LIN {X 0,Y 385.624,Z 461.843,A -85,B 0,C 180,E1 17447.458,E2 17447.458} C_VEL
LIN {X 0,Y 393.74,Z 473.597,A -85,B 0,C 180,E1 17445.289,E2 17445.289} C_VEL
LIN {X 0,Y 402.693,Z 487.716,A -85,B 0,C 180,E1 17443.13,E2 17443.13} C_VEL
LIN {X 0,Y 410.584,Z 501.659,A -85,B 0,C 180,E1 17441.371,E2 17441.371} C_VEL
LIN {X 0,Y 399.515,Z 724.653,A -85,B 0,C 180,E1 17436.869,E2 17436.869} C_VEL
LIN {X 0,Y 397.719,Z 745.499,A -85,B 0,C 180,E1 17436.196,E2 17436.196} C_VEL
LIN {X 0,Y 395.346,Z 765.584,A -85,B 0,C 180,E1 17435.296,E2 17435.296} C_VEL
LIN {X 0,Y 392.457,Z 785.369,A -85,B 0,C 180,E1 17434.136,E2 17434.136} C_VEL
LIN {X 0,Y 389.149,Z 804.356,A -85,B 0,C 180,E1 17432.737,E2 17432.737} C_VEL
LIN {X 0,Y 385.5,Z 822.639,A -85,B 0,C 180,E1 17431.079,E2 17431.079} C_VEL
LIN {X 0,Y 381.768,Z 839.649,A -85,B 0,C 180,E1 17429.2,E2 17429.2} C_VEL
LIN {X 0,Y 378.016,Z 855.337,A -85,B 0,C 180,E1 17427.11,E2 17427.11} C_VEL
LIN {X 0,Y 374.362,Z 870.021,A -85,B 0,C 180,E1 17424.767,E2 17424.767} C_VEL
LIN {X 0,Y 370.795,Z 884.125,A -85,B 0,C 180,E1 17422.061,E2 17422.061} C_VEL
LIN {X 0,Y 367.789,Z 896.136,A -85,B 0,C 180,E1 17419.272,E2 17419.272} C_VEL
LIN {X 0,Y 365.351,Z 906.362,A -85,B 0,C 180,E1 17416.397,E2 17416.397} C_VEL
LIN {X 0,Y 363.362,Z 915.457,A -85,B 0,C 180,E1 17413.243,E2 17413.243} C_VEL
LIN {X 0,Y 361.969,Z 922.647,A -85,B 0,C 180,E1 17410.056,E2 17410.056} C_VEL
LIN {X 0,Y 361.097,Z 928.123,A -85,B 0,C 180,E1 17406.848,E2 17406.848} C_VEL
LIN {X 0,Y 360.609,Z 932.126,A -85,B 0,C 180,E1 17403.483,E2 17403.483} C_VEL
LIN {X 0,Y 360.394,Z 934.36,A -85,B 0,C 180,E1 17400.322,E2 17400.322} C_VEL
LIN {X 0,Y 360.332,Z 935.093,A -85,B 0,C 180,E1 17397.243,E2 17397.243} C_VEL
LIN {X 0,Y 360.36,Z 934.348,A -85,B 0,C 180,E1 17394.066,E2 17394.066} C_VEL
LIN {X 0,Y 360.529,Z 932.047,A -85,B 0,C 180,E1 17390.788,E2 17390.788} C_VEL
LIN {X 0,Y 360.933,Z 928.226,A -85,B 0,C 180,E1 17387.571,E2 17387.571} C_VEL
LIN {X 0,Y 361.721,Z 922.518,A -85,B 0,C 180,E1 17384.238,E2 17384.238} C_VEL
LIN {X 0,Y 363.027,Z 914.958,A -85,B 0,C 180,E1 17380.951,E2 17380.951} C_VEL
LIN {X 0,Y 364.829,Z 905.967,A -85,B 0,C 180,E1 17377.872,E2 17377.872} C_VEL
LIN {X 0,Y 365.782,Z 901.545,A -85,B 0,C 180,E1 17376.571,E2 17376.571} C_VEL
LIN {X 0,Y 365.685,Z 897.934,A -85,B 0,C 180,E1 17375.494,E2 17375.494} C_VEL
LIN {X 0,Y 362.411,Z 888.671,A -85,B 0,C 180,E1 17372.727,E2 17372.727} C_VEL
LIN {X 0,Y 362.563,Z 884.364,A -85,B 0,C 180,E1 17371.705,E2 17371.705} C_VEL
LIN {X 0,Y 365.958,Z 870.807,A -85,B 0,C 180,E1 17369.057,E2 17369.057} C_VEL
LIN {X 0,Y 369.577,Z 856.128,A -85,B 0,C 180,E1 17366.665,E2 17366.665} C_VEL
LIN {X 0,Y 373.549,Z 839.227,A -85,B 0,C 180,E1 17364.39,E2 17364.39} C_VEL
LIN {X 0,Y 377.305,Z 821.832,A -85,B 0,C 180,E1 17362.459,E2 17362.459} C_VEL
LIN {X 0,Y 380.805,Z 804.113,A -85,B 0,C 180,E1 17360.841,E2 17360.841} C_VEL
LIN {X 0,Y 384.175,Z 784.574,A -85,B 0,C 180,E1 17359.386,E2 17359.386} C_VEL
LIN {X 0,Y 387.031,Z 764.817,A -85,B 0,C 180,E1 17358.221,E2 17358.221} C_VEL
LIN {X 0,Y 389.427,Z 744.323,A -85,B 0,C 180,E1 17357.301,E2 17357.301} C_VEL
LIN {X 0,Y 391.197,Z 723.212,A -85,B 0,C 180,E1 17356.623,E2 17356.623} C_VEL
LIN {X 0,Y 394.489,Z 650.13,A -85,B 0,C 180,E1 17355.144,E2 17355.144} C_VEL
LIN {X 0,Y 401.065,Z 502.372,A -85,B 0,C 180,E1 17352.239,E2 17352.239} C_VEL
LIN {X 0,Y 390.659,Z 484.683,A -85,B 0,C 180,E1 17350.151,E2 17350.151} C_VEL
LIN {X 0,Y 380.819,Z 469.313,A -85,B 0,C 180,E1 17348.046,E2 17348.046} C_VEL
LIN {X 0,Y 369.494,Z 452.63,A -85,B 0,C 180,E1 17345.369,E2 17345.369} C_VEL
LIN {X 0,Y 363.337,Z 440.093,A -85,B 0,C 180,E1 17342.05,E2 17342.05} C_VEL
LIN {X 0,Y 360.294,Z 434.531,A -85,B 0,C 180,E1 17340.395,E2 17340.395} C_VEL
LIN {X 0,Y 358.363,Z 430.7,A -85,B 0,C 180,E1 17339.244,E2 17339.244} C_VEL
LIN {X 0,Y 356.284,Z 426.499,A -85,B 0,C 180,E1 17337.944,E2 17337.944} C_VEL
LIN {X 0,Y 354.253,Z 423.304,A -85,B 0,C 180,E1 17336.798,E2 17336.798} C_VEL
LIN {X 0,Y 353.891,Z 421.837,A -85,B 0,C 180,E1 17336.274,E2 17336.274} C_VEL
LIN {X 0,Y 353.868,Z 421.638,A -85,B 0,C 180,E1 17332.029,E2 17332.029} C_VEL
LIN {X 0,Y 353.865,Z 421.638,A -85,B 0,C 180,E1 17327.738,E2 17327.738} C_VEL
LIN {X 0,Y 353.864,Z 421.647,A -85,B 0,C 180,E1 17323.431,E2 17323.431} C_VEL
LIN {X 0,Y 353.871,Z 421.657,A -85,B 0,C 180,E1 17319.266,E2 17319.266} C_VEL
LIN {X 0,Y 353.861,Z 421.644,A -85,B 0,C 180,E1 17314.97,E2 17314.97} C_VEL
LIN {X 0,Y 353.86,Z 421.627,A -85,B 0,C 180,E1 17310.76,E2 17310.76} C_VEL
LIN {X 0,Y 353.862,Z 421.627,A -85,B 0,C 180,E1 17306.697,E2 17306.697} C_VEL
LIN {X 0,Y 353.865,Z 421.651,A -85,B 0,C 180,E1 17302.424,E2 17302.424} C_VEL
LIN {X 0,Y 353.863,Z 421.647,A -85,B 0,C 180,E1 17298.109,E2 17298.109} C_VEL
LIN {X 0,Y 353.86,Z 421.626,A -85,B 0,C 180,E1 17293.897,E2 17293.897} C_VEL
LIN {X 0,Y 353.86,Z 421.63,A -85,B 0,C 180,E1 17289.761,E2 17289.761} C_VEL
LIN {X 0,Y 353.863,Z 421.653,A -85,B 0,C 180,E1 17285.513,E2 17285.513} C_VEL
LIN {X 0,Y 353.866,Z 421.645,A -85,B 0,C 180,E1 17281.296,E2 17281.296} C_VEL
LIN {X 0,Y 353.86,Z 421.629,A -85,B 0,C 180,E1 17277.085,E2 17277.085} C_VEL
LIN {X 0,Y 353.87,Z 421.625,A -85,B 0,C 180,E1 17272.859,E2 17272.859} C_VEL
LIN {X 0,Y 353.862,Z 421.633,A -85,B 0,C 180,E1 17268.593,E2 17268.593} C_VEL
LIN {X 0,Y 353.867,Z 421.64,A -85,B 0,C 180,E1 17264.43,E2 17264.43} C_VEL
LIN {X 0,Y 353.863,Z 421.642,A -85,B 0,C 180,E1 17260.181,E2 17260.181} C_VEL
LIN {X 0,Y 353.907,Z 421.916,A -85,B 0,C 180,E1 17256.647,E2 17256.647} C_VEL
LIN {X 0,Y 355.277,Z 425.289,A -85,B 0,C 180,E1 17255.563,E2 17255.563} C_VEL
LIN {X 0,Y 356.837,Z 427.334,A -85,B 0,C 180,E1 17254.793,E2 17254.793} C_VEL
LIN {X 0,Y 358.714,Z 431.017,A -85,B 0,C 180,E1 17253.693,E2 17253.693} C_VEL
LIN {X 0,Y 359.897,Z 433.003,A -85,B 0,C 180,E1 17253.074,E2 17253.074} C_VEL
LIN {X 0,Y 362.824,Z 438.361,A -85,B 0,C 180,E1 17251.527,E2 17251.527} C_VEL
LIN {X 0,Y 367.452,Z 446.794,A -85,B 0,C 180,E1 17249.233,E2 17249.233} C_VEL
LIN {X 0,Y 371.993,Z 455.21,A -85,B 0,C 180,E1 17247.208,E2 17247.208} C_VEL
LIN {X 0,Y 385.078,Z 473.968,A -85,B 0,C 180,E1 17244.207,E2 17244.207} C_VEL
LIN {X 0,Y 396.972,Z 492.362,A -85,B 0,C 180,E1 17241.713,E2 17241.713} C_VEL
LIN {X 0,Y 405.843,Z 507.315,A -85,B 0,C 180,E1 17239.976,E2 17239.976} C_VEL
LIN {X 0,Y 396.961,Z 726.559,A -85,B 0,C 180,E1 17235.789,E2 17235.789} C_VEL
LIN {X 0,Y 395.432,Z 758.529,A -85,B 0,C 180,E1 17235.13,E2 17235.13} C_VEL
LIN {X 0,Y 393.317,Z 780.529,A -85,B 0,C 180,E1 17234.471,E2 17234.471} C_VEL
LIN {X 0,Y 390.557,Z 801.649,A -85,B 0,C 180,E1 17233.573,E2 17233.573} C_VEL
LIN {X 0,Y 387.183,Z 823.142,A -85,B 0,C 180,E1 17232.379,E2 17232.379} C_VEL
LIN {X 0,Y 383.567,Z 842.972,A -85,B 0,C 180,E1 17231,E2 17231} C_VEL
LIN {X 0,Y 379.663,Z 861.754,A -85,B 0,C 180,E1 17229.399,E2 17229.399} C_VEL
LIN {X 0,Y 375.513,Z 880.297,A -85,B 0,C 180,E1 17227.49,E2 17227.49} C_VEL
LIN {X 0,Y 371.385,Z 897.84,A -85,B 0,C 180,E1 17225.339,E2 17225.339} C_VEL
LIN {X 0,Y 367.337,Z 914.388,A -85,B 0,C 180,E1 17222.927,E2 17222.927} C_VEL
LIN {X 0,Y 363.625,Z 929.506,A -85,B 0,C 180,E1 17220.3,E2 17220.3} C_VEL
LIN {X 0,Y 360.131,Z 944.253,A -85,B 0,C 180,E1 17217.268,E2 17217.268} C_VEL
LIN {X 0,Y 357.383,Z 956.769,A -85,B 0,C 180,E1 17214.21,E2 17214.21} C_VEL
LIN {X 0,Y 355.303,Z 967.347,A -85,B 0,C 180,E1 17211.116,E2 17211.116} C_VEL
LIN {X 0,Y 353.742,Z 976.8,A -85,B 0,C 180,E1 17207.777,E2 17207.777} C_VEL
LIN {X 0,Y 352.792,Z 984.497,A -85,B 0,C 180,E1 17204.445,E2 17204.445} C_VEL
LIN {X 0,Y 352.315,Z 990.433,A -85,B 0,C 180,E1 17201.13,E2 17201.13} C_VEL
LIN {X 0,Y 352.13,Z 994.962,A -85,B 0,C 180,E1 17197.673,E2 17197.673} C_VEL
LIN {X 0,Y 352.135,Z 997.53,A -85,B 0,C 180,E1 17194.706,E2 17194.706} C_VEL
LIN {X 0,Y 352.185,Z 998.914,A -85,B 0,C 180,E1 17191.305,E2 17191.305} C_VEL
LIN {X 0,Y 352.184,Z 998.823,A -85,B 0,C 180,E1 17188.377,E2 17188.377} C_VEL
LIN {X 0,Y 352.141,Z 997.271,A -85,B 0,C 180,E1 17185.117,E2 17185.117} C_VEL
LIN {X 0,Y 352.148,Z 994.589,A -85,B 0,C 180,E1 17182.171,E2 17182.171} C_VEL
LIN {X 0,Y 352.34,Z 989.877,A -85,B 0,C 180,E1 17178.712,E2 17178.712} C_VEL
LIN {X 0,Y 352.825,Z 983.792,A -85,B 0,C 180,E1 17175.395,E2 17175.395} C_VEL
LIN {X 0,Y 353.789,Z 975.895,A -85,B 0,C 180,E1 17172.062,E2 17172.062} C_VEL
LIN {X 0,Y 355.462,Z 965.704,A -85,B 0,C 180,E1 17168.556,E2 17168.556} C_VEL
LIN {X 0,Y 357.648,Z 954.623,A -85,B 0,C 180,E1 17165.388,E2 17165.388} C_VEL
LIN {X 0,Y 360.561,Z 941.345,A -85,B 0,C 180,E1 17162.238,E2 17162.238} C_VEL
LIN {X 0,Y 363.858,Z 927.441,A -85,B 0,C 180,E1 17159.45,E2 17159.45} C_VEL
LIN {X 0,Y 367.695,Z 911.791,A -85,B 0,C 180,E1 17156.78,E2 17156.78} C_VEL
LIN {X 0,Y 371.908,Z 894.648,A -85,B 0,C 180,E1 17154.316,E2 17154.316} C_VEL
LIN {X 0,Y 376.215,Z 876.414,A -85,B 0,C 180,E1 17152.132,E2 17152.132} C_VEL
LIN {X 0,Y 380.472,Z 857.446,A -85,B 0,C 180,E1 17150.236,E2 17150.236} C_VEL
LIN {X 0,Y 384.412,Z 838.439,A -85,B 0,C 180,E1 17148.656,E2 17148.656} C_VEL
LIN {X 0,Y 387.995,Z 818.936,A -85,B 0,C 180,E1 17147.338,E2 17147.338} C_VEL
LIN {X 0,Y 391.235,Z 798.45,A -85,B 0,C 180,E1 17146.233,E2 17146.233} C_VEL
LIN {X 0,Y 394.042,Z 777.211,A -85,B 0,C 180,E1 17145.357,E2 17145.357} C_VEL
LIN {X 0,Y 396.122,Z 755.661,A -85,B 0,C 180,E1 17144.721,E2 17144.721} C_VEL
LIN {X 0,Y 397.895,Z 717.515,A -85,B 0,C 180,E1 17143.948,E2 17143.948} C_VEL
LIN {X 0,Y 406.806,Z 512.285,A -85,B 0,C 180,E1 17139.967,E2 17139.967} C_VEL
LIN {X 0,Y 406.945,Z 506.851,A -85,B 0,C 180,E1 17139.84,E2 17139.84} C_VEL
LIN {X 0,Y 398.811,Z 492.533,A -85,B 0,C 180,E1 17138.01,E2 17138.01} C_VEL
LIN {X 0,Y 390.411,Z 479.057,A -85,B 0,C 180,E1 17135.952,E2 17135.952} C_VEL
LIN {X 0,Y 381.877,Z 466.595,A -85,B 0,C 180,E1 17133.625,E2 17133.625} C_VEL
LIN {X 0,Y 374.629,Z 456.983,A -85,B 0,C 180,E1 17131.406,E2 17131.406} C_VEL
LIN {X 0,Y 372.382,Z 453.459,A -85,B 0,C 180,E1 17130.495,E2 17130.495} C_VEL
LIN {X 0,Y 369.247,Z 447.902,A -85,B 0,C 180,E1 17128.462,E2 17128.462} C_VEL
LIN {X 0,Y 366.715,Z 443.261,A -85,B 0,C 180,E1 17126.56,E2 17126.56} C_VEL
LIN {X 0,Y 364.44,Z 439.225,A -85,B 0,C 180,E1 17124.646,E2 17124.646} C_VEL
LIN {X 0,Y 361.343,Z 434.166,A -85,B 0,C 180,E1 17121.593,E2 17121.593} C_VEL
LIN {X 0,Y 360.702,Z 432.95,A -85,B 0,C 180,E1 17120.782,E2 17120.782} C_VEL
LIN {X 0,Y 357.518,Z 427.654,A -85,B 0,C 180,E1 17115.075,E2 17115.075} C_VEL
LIN {X 0,Y 356.711,Z 426.904,A -85,B 0,C 180,E1 17110.988,E2 17110.988} C_VEL
LIN {X 0,Y 357.579,Z 427.797,A -85,B 0,C 180,E1 17106.905,E2 17106.905} C_VEL
LIN {X 0,Y 361.007,Z 433.575,A -85,B 0,C 180,E1 17100.952,E2 17100.952} C_VEL
LIN {X 0,Y 363.131,Z 437.618,A -85,B 0,C 180,E1 17098.422,E2 17098.422} C_VEL
LIN {X 0,Y 364.003,Z 438.907,A -85,B 0,C 180,E1 17097.638,E2 17097.638} C_VEL
LIN {X 0,Y 366.024,Z 442.707,A -85,B 0,C 180,E1 17095.77,E2 17095.77} C_VEL
LIN {X 0,Y 366.893,Z 444.481,A -85,B 0,C 180,E1 17094.997,E2 17094.997} C_VEL
LIN {X 0,Y 369.261,Z 448.859,A -85,B 0,C 180,E1 17093.157,E2 17093.157} C_VEL
LIN {X 0,Y 371.755,Z 453.713,A -85,B 0,C 180,E1 17091.415,E2 17091.415} C_VEL
LIN {X 0,Y 378.963,Z 463.457,A -85,B 0,C 180,E1 17089.01,E2 17089.01} C_VEL
LIN {X 0,Y 385.61,Z 472.854,A -85,B 0,C 180,E1 17087.061,E2 17087.061} C_VEL
LIN {X 0,Y 394.091,Z 485.886,A -85,B 0,C 180,E1 17084.813,E2 17084.813} C_VEL
LIN {X 0,Y 402.845,Z 500.747,A -85,B 0,C 180,E1 17082.709,E2 17082.709} C_VEL
LIN {X 0,Y 405.224,Z 505.329,A -85,B 0,C 180,E1 17082.16,E2 17082.16} C_VEL
LIN {X 0,Y 393.777,Z 725.022,A -85,B 0,C 180,E1 17077.674,E2 17077.674} C_VEL
LIN {X 0,Y 391.902,Z 745.893,A -85,B 0,C 180,E1 17076.993,E2 17076.993} C_VEL
LIN {X 0,Y 389.528,Z 765.225,A -85,B 0,C 180,E1 17076.123,E2 17076.123} C_VEL
LIN {X 0,Y 386.385,Z 785.898,A -85,B 0,C 180,E1 17074.907,E2 17074.907} C_VEL
LIN {X 0,Y 383.048,Z 804.359,A -85,B 0,C 180,E1 17073.539,E2 17073.539} C_VEL
LIN {X 0,Y 379.303,Z 822.416,A -85,B 0,C 180,E1 17071.898,E2 17071.898} C_VEL
LIN {X 0,Y 375.129,Z 840.491,A -85,B 0,C 180,E1 17069.878,E2 17069.878} C_VEL
LIN {X 0,Y 371.183,Z 856.196,A -85,B 0,C 180,E1 17067.751,E2 17067.751} C_VEL
LIN {X 0,Y 367.371,Z 870.732,A -85,B 0,C 180,E1 17065.394,E2 17065.394} C_VEL
LIN {X 0,Y 363.788,Z 884.115,A -85,B 0,C 180,E1 17062.795,E2 17062.795} C_VEL
LIN {X 0,Y 360.755,Z 895.549,A -85,B 0,C 180,E1 17060.143,E2 17060.143} C_VEL
LIN {X 0,Y 357.936,Z 906.576,A -85,B 0,C 180,E1 17057.031,E2 17057.031} C_VEL
LIN {X 0,Y 355.716,Z 915.92,A -85,B 0,C 180,E1 17053.74,E2 17053.74} C_VEL
LIN {X 0,Y 354.193,Z 923.167,A -85,B 0,C 180,E1 17050.481,E2 17050.481} C_VEL
LIN {X 0,Y 353.242,Z 928.592,A -85,B 0,C 180,E1 17047.276,E2 17047.276} C_VEL
LIN {X 0,Y 352.704,Z 932.594,A -85,B 0,C 180,E1 17043.944,E2 17043.944} C_VEL
LIN {X 0,Y 352.451,Z 934.981,A -85,B 0,C 180,E1 17040.701,E2 17040.701} C_VEL
LIN {X 0,Y 352.365,Z 935.784,A -85,B 0,C 180,E1 17037.545,E2 17037.545} C_VEL
LIN {X 0,Y 352.39,Z 935.18,A -85,B 0,C 180,E1 17034.289,E2 17034.289} C_VEL
LIN {X 0,Y 352.54,Z 933.159,A -85,B 0,C 180,E1 17031.076,E2 17031.076} C_VEL
LIN {X 0,Y 352.941,Z 929.545,A -85,B 0,C 180,E1 17027.812,E2 17027.812} C_VEL
LIN {X 0,Y 353.672,Z 924.319,A -85,B 0,C 180,E1 17024.569,E2 17024.569} C_VEL
LIN {X 0,Y 354.901,Z 917.473,A -85,B 0,C 180,E1 17021.356,E2 17021.356} C_VEL
LIN {X 0,Y 356.67,Z 908.995,A -85,B 0,C 180,E1 17018.216,E2 17018.216} C_VEL
LIN {X 0,Y 358.942,Z 899.215,A -85,B 0,C 180,E1 17015.271,E2 17015.271} C_VEL
LIN {X 0,Y 361.991,Z 886.756,A -85,B 0,C 180,E1 17012.213,E2 17012.213} C_VEL
LIN {X 0,Y 362.563,Z 884.364,A -85,B 0,C 180,E1 17011.705,E2 17011.705} C_VEL
LIN {X 0,Y 362.794,Z 879.981,A -85,B 0,C 180,E1 17010.698,E2 17010.698} C_VEL
LIN {X 0,Y 360.416,Z 868.807,A -85,B 0,C 180,E1 17008.065,E2 17008.065} C_VEL
LIN {X 0,Y 360.833,Z 863.748,A -85,B 0,C 180,E1 17007.134,E2 17007.134} C_VEL
LIN {X 0,Y 364.759,Z 848.234,A -85,B 0,C 180,E1 17004.807,E2 17004.807} C_VEL
LIN {X 0,Y 368.832,Z 831.005,A -85,B 0,C 180,E1 17002.677,E2 17002.677} C_VEL
LIN {X 0,Y 372.614,Z 813.432,A -85,B 0,C 180,E1 17000.888,E2 17000.888} C_VEL
LIN {X 0,Y 376.151,Z 795.04,A -85,B 0,C 180,E1 16999.351,E2 16999.351} C_VEL
LIN {X 0,Y 379.348,Z 775.813,A -85,B 0,C 180,E1 16998.056,E2 16998.056} C_VEL
LIN {X 0,Y 382.057,Z 756.052,A -85,B 0,C 180,E1 16997.01,E2 16997.01} C_VEL
LIN {X 0,Y 384.301,Z 734.61,A -85,B 0,C 180,E1 16996.167,E2 16996.167} C_VEL
LIN {X 0,Y 385.812,Z 712.602,A -85,B 0,C 180,E1 16995.591,E2 16995.591} C_VEL
LIN {X 0,Y 395.371,Z 505.74,A -85,B 0,C 180,E1 16991.473,E2 16991.473} C_VEL
LIN {X 0,Y 384.405,Z 487.101,A -85,B 0,C 180,E1 16989.19,E2 16989.19} C_VEL
LIN {X 0,Y 373.707,Z 470.564,A -85,B 0,C 180,E1 16986.787,E2 16986.787} C_VEL
LIN {X 0,Y 362.79,Z 454.87,A -85,B 0,C 180,E1 16984.119,E2 16984.119} C_VEL
LIN {X 0,Y 360.902,Z 451.951,A -85,B 0,C 180,E1 16983.491,E2 16983.491} C_VEL
LIN {X 0,Y 355.739,Z 441.48,A -85,B 0,C 180,E1 16980.534,E2 16980.534} C_VEL
LIN {X 0,Y 352.83,Z 436.157,A -85,B 0,C 180,E1 16978.851,E2 16978.851} C_VEL
LIN {X 0,Y 350.758,Z 432.078,A -85,B 0,C 180,E1 16977.541,E2 16977.541} C_VEL
LIN {X 0,Y 348.747,Z 428.234,A -85,B 0,C 180,E1 16976.247,E2 16976.247} C_VEL
LIN {X 0,Y 346.289,Z 424.207,A -85,B 0,C 180,E1 16974.724,E2 16974.724} C_VEL
LIN {X 0,Y 345.952,Z 422.807,A -85,B 0,C 180,E1 16974.176,E2 16974.176} C_VEL
LIN {X 0,Y 345.929,Z 422.624,A -85,B 0,C 180,E1 16969.992,E2 16969.992} C_VEL
LIN {X 0,Y 345.924,Z 422.619,A -85,B 0,C 180,E1 16965.793,E2 16965.793} C_VEL
LIN {X 0,Y 345.93,Z 422.614,A -85,B 0,C 180,E1 16961.527,E2 16961.527} C_VEL
LIN {X 0,Y 345.923,Z 422.617,A -85,B 0,C 180,E1 16957.354,E2 16957.354} C_VEL
LIN {X 0,Y 345.927,Z 422.633,A -85,B 0,C 180,E1 16953.045,E2 16953.045} C_VEL
LIN {X 0,Y 345.931,Z 422.643,A -85,B 0,C 180,E1 16948.859,E2 16948.859} C_VEL
LIN {X 0,Y 345.921,Z 422.618,A -85,B 0,C 180,E1 16944.597,E2 16944.597} C_VEL
LIN {X 0,Y 345.922,Z 422.611,A -85,B 0,C 180,E1 16940.472,E2 16940.472} C_VEL
LIN {X 0,Y 345.924,Z 422.633,A -85,B 0,C 180,E1 16936.283,E2 16936.283} C_VEL
LIN {X 0,Y 345.924,Z 422.644,A -85,B 0,C 180,E1 16932.012,E2 16932.012} C_VEL
LIN {X 0,Y 345.924,Z 422.619,A -85,B 0,C 180,E1 16927.641,E2 16927.641} C_VEL
LIN {X 0,Y 345.92,Z 422.61,A -85,B 0,C 180,E1 16923.48,E2 16923.48} C_VEL
LIN {X 0,Y 345.927,Z 422.623,A -85,B 0,C 180,E1 16919.172,E2 16919.172} C_VEL
LIN {X 0,Y 345.926,Z 422.644,A -85,B 0,C 180,E1 16914.86,E2 16914.86} C_VEL
LIN {X 0,Y 345.927,Z 422.641,A -85,B 0,C 180,E1 16910.686,E2 16910.686} C_VEL
LIN {X 0,Y 345.926,Z 422.629,A -85,B 0,C 180,E1 16906.461,E2 16906.461} C_VEL
LIN {X 0,Y 345.921,Z 422.627,A -85,B 0,C 180,E1 16902.159,E2 16902.159} C_VEL
LIN {X 0,Y 345.972,Z 422.927,A -85,B 0,C 180,E1 16898.763,E2 16898.763} C_VEL
LIN {X 0,Y 347.562,Z 426.583,A -85,B 0,C 180,E1 16897.505,E2 16897.505} C_VEL
LIN {X 0,Y 349.033,Z 428.574,A -85,B 0,C 180,E1 16896.714,E2 16896.714} C_VEL
LIN {X 0,Y 351.155,Z 432.409,A -85,B 0,C 180,E1 16895.436,E2 16895.436} C_VEL
LIN {X 0,Y 352.235,Z 434.417,A -85,B 0,C 180,E1 16894.8,E2 16894.8} C_VEL
LIN {X 0,Y 354.806,Z 438.879,A -85,B 0,C 180,E1 16893.381,E2 16893.381} C_VEL
LIN {X 0,Y 359.813,Z 448.064,A -85,B 0,C 180,E1 16890.721,E2 16890.721} C_VEL
LIN {X 0,Y 363.635,Z 455.167,A -85,B 0,C 180,E1 16888.92,E2 16888.92} C_VEL
LIN {X 0,Y 372.943,Z 468.041,A -85,B 0,C 180,E1 16886.615,E2 16886.615} C_VEL
LIN {X 0,Y 384.43,Z 484.99,A -85,B 0,C 180,E1 16883.999,E2 16883.999} C_VEL
LIN {X 0,Y 396.178,Z 503.807,A -85,B 0,C 180,E1 16881.53,E2 16881.53} C_VEL
LIN {X 0,Y 400.156,Z 510.945,A -85,B 0,C 180,E1 16880.731,E2 16880.731} C_VEL
LIN {X 0,Y 390.768,Z 732.765,A -85,B 0,C 180,E1 16876.451,E2 16876.451} C_VEL
LIN {X 0,Y 389.222,Z 760.597,A -85,B 0,C 180,E1 16875.846,E2 16875.846} C_VEL
LIN {X 0,Y 386.976,Z 782.262,A -85,B 0,C 180,E1 16875.166,E2 16875.166} C_VEL
LIN {X 0,Y 384.094,Z 803.402,A -85,B 0,C 180,E1 16874.241,E2 16874.241} C_VEL
LIN {X 0,Y 380.698,Z 823.875,A -85,B 0,C 180,E1 16873.07,E2 16873.07} C_VEL
LIN {X 0,Y 376.885,Z 843.783,A -85,B 0,C 180,E1 16871.652,E2 16871.652} C_VEL
LIN {X 0,Y 372.727,Z 862.989,A -85,B 0,C 180,E1 16869.979,E2 16869.979} C_VEL
LIN {X 0,Y 368.404,Z 881.303,A -85,B 0,C 180,E1 16868.033,E2 16868.033} C_VEL
LIN {X 0,Y 363.951,Z 899.231,A -85,B 0,C 180,E1 16865.759,E2 16865.759} C_VEL
LIN {X 0,Y 359.762,Z 915.586,A -85,B 0,C 180,E1 16863.294,E2 16863.294} C_VEL
LIN {X 0,Y 355.873,Z 930.758,A -85,B 0,C 180,E1 16860.569,E2 16860.569} C_VEL
LIN {X 0,Y 352.526,Z 944.114,A -85,B 0,C 180,E1 16857.723,E2 16857.723} C_VEL
LIN {X 0,Y 349.566,Z 956.872,A -85,B 0,C 180,E1 16854.506,E2 16854.506} C_VEL
LIN {X 0,Y 347.281,Z 968.073,A -85,B 0,C 180,E1 16851.121,E2 16851.121} C_VEL
LIN {X 0,Y 345.697,Z 977.308,A -85,B 0,C 180,E1 16847.683,E2 16847.683} C_VEL
LIN {X 0,Y 344.728,Z 985.032,A -85,B 0,C 180,E1 16844.104,E2 16844.104} C_VEL
LIN {X 0,Y 344.287,Z 990.748,A -85,B 0,C 180,E1 16840.715,E2 16840.715} C_VEL
LIN {X 0,Y 344.143,Z 994.746,A -85,B 0,C 180,E1 16837.348,E2 16837.348} C_VEL
LIN {X 0,Y 344.18,Z 997.304,A -85,B 0,C 180,E1 16834.001,E2 16834.001} C_VEL
LIN {X 0,Y 344.212,Z 998.266,A -85,B 0,C 180,E1 16830.836,E2 16830.836} C_VEL
LIN {X 0,Y 344.195,Z 997.88,A -85,B 0,C 180,E1 16827.506,E2 16827.506} C_VEL
LIN {X 0,Y 344.171,Z 996.05,A -85,B 0,C 180,E1 16824.335,E2 16824.335} C_VEL
LIN {X 0,Y 344.207,Z 992.485,A -85,B 0,C 180,E1 16820.811,E2 16820.811} C_VEL
LIN {X 0,Y 344.459,Z 987.755,A -85,B 0,C 180,E1 16817.6,E2 16817.6} C_VEL
LIN {X 0,Y 345.163,Z 980.805,A -85,B 0,C 180,E1 16814.031,E2 16814.031} C_VEL
LIN {X 0,Y 346.381,Z 972.477,A -85,B 0,C 180,E1 16810.617,E2 16810.617} C_VEL
LIN {X 0,Y 348.277,Z 962.186,A -85,B 0,C 180,E1 16807.201,E2 16807.201} C_VEL
LIN {X 0,Y 350.813,Z 950.478,A -85,B 0,C 180,E1 16803.97,E2 16803.97} C_VEL
LIN {X 0,Y 353.944,Z 937.466,A -85,B 0,C 180,E1 16800.935,E2 16800.935} C_VEL
LIN {X 0,Y 357.589,Z 923.081,A -85,B 0,C 180,E1 16798.103,E2 16798.103} C_VEL
LIN {X 0,Y 361.71,Z 907.131,A -85,B 0,C 180,E1 16795.461,E2 16795.461} C_VEL
LIN {X 0,Y 366.327,Z 889.13,A -85,B 0,C 180,E1 16792.955,E2 16792.955} C_VEL
LIN {X 0,Y 370.733,Z 871.292,A -85,B 0,C 180,E1 16790.875,E2 16790.875} C_VEL
LIN {X 0,Y 375.132,Z 852.283,A -85,B 0,C 180,E1 16789.035,E2 16789.035} C_VEL
LIN {X 0,Y 379.255,Z 832.565,A -85,B 0,C 180,E1 16787.472,E2 16787.472} C_VEL
LIN {X 0,Y 383.215,Z 811.153,A -85,B 0,C 180,E1 16786.108,E2 16786.108} C_VEL
LIN {X 0,Y 386.468,Z 790.424,A -85,B 0,C 180,E1 16785.072,E2 16785.072} C_VEL
LIN {X 0,Y 389.098,Z 769.004,A -85,B 0,C 180,E1 16784.282,E2 16784.282} C_VEL
LIN {X 0,Y 390.946,Z 746.701,A -85,B 0,C 180,E1 16783.702,E2 16783.702} C_VEL
LIN {X 0,Y 401.06,Z 524.263,A -85,B 0,C 180,E1 16779.334,E2 16779.334} C_VEL
LIN {X 0,Y 401.64,Z 510.251,A -85,B 0,C 180,E1 16779.037,E2 16779.037} C_VEL
LIN {X 0,Y 393.173,Z 495.407,A -85,B 0,C 180,E1 16777.033,E2 16777.033} C_VEL
LIN {X 0,Y 384.226,Z 481.128,A -85,B 0,C 180,E1 16774.691,E2 16774.691} C_VEL
LIN {X 0,Y 376.015,Z 469.255,A -85,B 0,C 180,E1 16772.267,E2 16772.267} C_VEL
LIN {X 0,Y 368.607,Z 459.454,A -85,B 0,C 180,E1 16769.761,E2 16769.761} C_VEL
LIN {X 0,Y 364.668,Z 454.303,A -85,B 0,C 180,E1 16768.227,E2 16768.227} C_VEL
LIN {X 0,Y 362.252,Z 449.817,A -85,B 0,C 180,E1 16766.383,E2 16766.383} C_VEL
LIN {X 0,Y 359.98,Z 445.622,A -85,B 0,C 180,E1 16764.364,E2 16764.364} C_VEL
LIN {X 0,Y 357.141,Z 441.049,A -85,B 0,C 180,E1 16761.515,E2 16761.515} C_VEL
LIN {X 0,Y 356.541,Z 439.764,A -85,B 0,C 180,E1 16760.692,E2 16760.692} C_VEL
LIN {X 0,Y 353.444,Z 434.523,A -85,B 0,C 180,E1 16754.917,E2 16754.917} C_VEL
LIN {X 0,Y 352.669,Z 433.82,A -85,B 0,C 180,E1 16750.784,E2 16750.784} C_VEL
LIN {X 0,Y 353.49,Z 434.698,A -85,B 0,C 180,E1 16746.916,E2 16746.916} C_VEL
LIN {X 0,Y 356.617,Z 440.194,A -85,B 0,C 180,E1 16741.124,E2 16741.124} C_VEL
LIN {X 0,Y 358.888,Z 444.434,A -85,B 0,C 180,E1 16738.403,E2 16738.403} C_VEL
LIN {X 0,Y 359.722,Z 446.282,A -85,B 0,C 180,E1 16737.451,E2 16737.451} C_VEL
LIN {X 0,Y 362.024,Z 450.324,A -85,B 0,C 180,E1 16735.406,E2 16735.406} C_VEL
LIN {X 0,Y 364.3,Z 454.251,A -85,B 0,C 180,E1 16733.736,E2 16733.736} C_VEL
LIN {X 0,Y 368.139,Z 459.291,A -85,B 0,C 180,E1 16732.234,E2 16732.234} C_VEL
LIN {X 0,Y 376.225,Z 470.464,A -85,B 0,C 180,E1 16729.433,E2 16729.433} C_VEL
LIN {X 0,Y 383.376,Z 480.863,A -85,B 0,C 180,E1 16727.276,E2 16727.276} C_VEL
LIN {X 0,Y 391.567,Z 493.917,A -85,B 0,C 180,E1 16725.054,E2 16725.054} C_VEL
LIN {X 0,Y 399.88,Z 508.388,A -85,B 0,C 180,E1 16723.008,E2 16723.008} C_VEL
LIN {X 0,Y 390.561,Z 681.077,A -85,B 0,C 180,E1 16719.453,E2 16719.453} C_VEL
LIN {X 0,Y 388.008,Z 726.793,A -85,B 0,C 180,E1 16718.462,E2 16718.462} C_VEL
LIN {X 0,Y 386.035,Z 747.663,A -85,B 0,C 180,E1 16717.765,E2 16717.765} C_VEL
LIN {X 0,Y 383.491,Z 767.196,A -85,B 0,C 180,E1 16716.86,E2 16716.86} C_VEL
LIN {X 0,Y 380.257,Z 787.34,A -85,B 0,C 180,E1 16715.645,E2 16715.645} C_VEL
LIN {X 0,Y 376.54,Z 806.697,A -85,B 0,C 180,E1 16714.17,E2 16714.17} C_VEL
LIN {X 0,Y 372.661,Z 824.354,A -85,B 0,C 180,E1 16712.517,E2 16712.517} C_VEL
LIN {X 0,Y 368.51,Z 841.55,A -85,B 0,C 180,E1 16710.559,E2 16710.559} C_VEL
LIN {X 0,Y 364.221,Z 857.792,A -85,B 0,C 180,E1 16708.312,E2 16708.312} C_VEL
LIN {X 0,Y 360.192,Z 872.296,A -85,B 0,C 180,E1 16705.893,E2 16705.893} C_VEL
LIN {X 0,Y 356.34,Z 885.903,A -85,B 0,C 180,E1 16703.167,E2 16703.167} C_VEL
LIN {X 0,Y 352.852,Z 898.26,A -85,B 0,C 180,E1 16700.16,E2 16700.16} C_VEL
LIN {X 0,Y 350.137,Z 908.297,A -85,B 0,C 180,E1 16697.184,E2 16697.184} C_VEL
LIN {X 0,Y 347.977,Z 916.929,A -85,B 0,C 180,E1 16694.048,E2 16694.048} C_VEL
LIN {X 0,Y 346.311,Z 924.355,A -85,B 0,C 180,E1 16690.594,E2 16690.594} C_VEL
LIN {X 0,Y 345.289,Z 929.779,A -85,B 0,C 180,E1 16687.219,E2 16687.219} C_VEL
LIN {X 0,Y 344.737,Z 933.579,A -85,B 0,C 180,E1 16683.834,E2 16683.834} C_VEL
LIN {X 0,Y 344.472,Z 935.834,A -85,B 0,C 180,E1 16680.45,E2 16680.45} C_VEL
LIN {X 0,Y 344.398,Z 936.548,A -85,B 0,C 180,E1 16677.112,E2 16677.112} C_VEL
LIN {X 0,Y 344.434,Z 935.704,A -85,B 0,C 180,E1 16673.793,E2 16673.793} C_VEL
LIN {X 0,Y 344.654,Z 933.312,A -85,B 0,C 180,E1 16670.368,E2 16670.368} C_VEL
LIN {X 0,Y 345.131,Z 929.408,A -85,B 0,C 180,E1 16667.01,E2 16667.01} C_VEL
LIN {X 0,Y 346.015,Z 923.963,A -85,B 0,C 180,E1 16663.703,E2 16663.703} C_VEL
LIN {X 0,Y 347.416,Z 916.817,A -85,B 0,C 180,E1 16660.442,E2 16660.442} C_VEL
LIN {X 0,Y 349.425,Z 907.942,A -85,B 0,C 180,E1 16657.229,E2 16657.229} C_VEL
LIN {X 0,Y 352.102,Z 897.143,A -85,B 0,C 180,E1 16654.067,E2 16654.067} C_VEL
LIN {X 0,Y 355.299,Z 884.864,A -85,B 0,C 180,E1 16651.125,E2 16651.125} C_VEL
LIN {X 0,Y 358.695,Z 872.001,A -85,B 0,C 180,E1 16648.559,E2 16648.559} C_VEL
LIN {X 0,Y 360.833,Z 863.748,A -85,B 0,C 180,E1 16647.134,E2 16647.134} C_VEL
LIN {X 0,Y 361.299,Z 858.618,A -85,B 0,C 180,E1 16646.225,E2 16646.225} C_VEL
LIN {X 0,Y 359.589,Z 845.6,A -85,B 0,C 180,E1 16643.791,E2 16643.791} C_VEL
LIN {X 0,Y 360.199,Z 839.917,A -85,B 0,C 180,E1 16642.955,E2 16642.955} C_VEL
LIN {X 0,Y 364.259,Z 822.619,A -85,B 0,C 180,E1 16640.995,E2 16640.995} C_VEL
LIN {X 0,Y 368.022,Z 804.981,A -85,B 0,C 180,E1 16639.351,E2 16639.351} C_VEL
LIN {X 0,Y 371.616,Z 785.67,A -85,B 0,C 180,E1 16637.883,E2 16637.883} C_VEL
LIN {X 0,Y 374.706,Z 765.908,A -85,B 0,C 180,E1 16636.691,E2 16636.691} C_VEL
LIN {X 0,Y 377.291,Z 745.454,A -85,B 0,C 180,E1 16635.751,E2 16635.751} C_VEL
LIN {X 0,Y 379.203,Z 724.319,A -85,B 0,C 180,E1 16635.056,E2 16635.056} C_VEL
LIN {X 0,Y 381.986,Z 668.708,A -85,B 0,C 180,E1 16633.891,E2 16633.891} C_VEL
LIN {X 0,Y 389.705,Z 509.047,A -85,B 0,C 180,E1 16630.682,E2 16630.682} C_VEL
LIN {X 0,Y 379.008,Z 490.937,A -85,B 0,C 180,E1 16628.374,E2 16628.374} C_VEL
LIN {X 0,Y 368.264,Z 474.237,A -85,B 0,C 180,E1 16625.868,E2 16625.868} C_VEL
LIN {X 0,Y 358.39,Z 460.064,A -85,B 0,C 180,E1 16623.356,E2 16623.356} C_VEL
LIN {X 0,Y 353.087,Z 452.669,A -85,B 0,C 180,E1 16621.87,E2 16621.87} C_VEL
LIN {X 0,Y 348.106,Z 442.756,A -85,B 0,C 180,E1 16618.865,E2 16618.865} C_VEL
LIN {X 0,Y 345.464,Z 437.884,A -85,B 0,C 180,E1 16617.23,E2 16617.23} C_VEL
LIN {X 0,Y 342.875,Z 433.094,A -85,B 0,C 180,E1 16615.544,E2 16615.544} C_VEL
LIN {X 0,Y 340.834,Z 429.01,A -85,B 0,C 180,E1 16614.073,E2 16614.073} C_VEL
LIN {X 0,Y 338.405,Z 425.361,A -85,B 0,C 180,E1 16612.505,E2 16612.505} C_VEL
LIN {X 0,Y 338.018,Z 423.817,A -85,B 0,C 180,E1 16611.891,E2 16611.891} C_VEL
LIN {X 0,Y 337.984,Z 423.612,A -85,B 0,C 180,E1 16607.582,E2 16607.582} C_VEL
LIN {X 0,Y 337.984,Z 423.619,A -85,B 0,C 180,E1 16603.299,E2 16603.299} C_VEL
LIN {X 0,Y 337.985,Z 423.633,A -85,B 0,C 180,E1 16598.916,E2 16598.916} C_VEL
LIN {X 0,Y 337.983,Z 423.627,A -85,B 0,C 180,E1 16594.611,E2 16594.611} C_VEL
LIN {X 0,Y 337.989,Z 423.607,A -85,B 0,C 180,E1 16590.193,E2 16590.193} C_VEL
LIN {X 0,Y 337.987,Z 423.597,A -85,B 0,C 180,E1 16585.927,E2 16585.927} C_VEL
LIN {X 0,Y 337.992,Z 423.612,A -85,B 0,C 180,E1 16581.702,E2 16581.702} C_VEL
LIN {X 0,Y 337.988,Z 423.633,A -85,B 0,C 180,E1 16577.385,E2 16577.385} C_VEL
LIN {X 0,Y 337.983,Z 423.613,A -85,B 0,C 180,E1 16572.993,E2 16572.993} C_VEL
LIN {X 0,Y 337.982,Z 423.599,A -85,B 0,C 180,E1 16568.678,E2 16568.678} C_VEL
LIN {X 0,Y 337.98,Z 423.607,A -85,B 0,C 180,E1 16564.412,E2 16564.412} C_VEL
LIN {X 0,Y 337.994,Z 423.627,A -85,B 0,C 180,E1 16560,E2 16560} C_VEL
LIN {X 0,Y 337.985,Z 423.632,A -85,B 0,C 180,E1 16555.543,E2 16555.543} C_VEL
LIN {X 0,Y 337.988,Z 423.618,A -85,B 0,C 180,E1 16551.15,E2 16551.15} C_VEL
LIN {X 0,Y 337.989,Z 423.613,A -85,B 0,C 180,E1 16546.73,E2 16546.73} C_VEL
LIN {X 0,Y 337.986,Z 423.611,A -85,B 0,C 180,E1 16542.438,E2 16542.438} C_VEL
LIN {X 0,Y 338.053,Z 424.043,A -85,B 0,C 180,E1 16541.063,E2 16541.063} C_VEL
LIN {X 0,Y 339.481,Z 427.374,A -85,B 0,C 180,E1 16539.843,E2 16539.843} C_VEL
LIN {X 0,Y 341.159,Z 429.546,A -85,B 0,C 180,E1 16538.871,E2 16538.871} C_VEL
LIN {X 0,Y 343.12,Z 433.269,A -85,B 0,C 180,E1 16537.559,E2 16537.559} C_VEL
LIN {X 0,Y 344.224,Z 434.975,A -85,B 0,C 180,E1 16536.913,E2 16536.913} C_VEL
LIN {X 0,Y 347.188,Z 440.308,A -85,B 0,C 180,E1 16535.12,E2 16535.12} C_VEL
LIN {X 0,Y 350.373,Z 446.193,A -85,B 0,C 180,E1 16533.283,E2 16533.283} C_VEL
LIN {X 0,Y 352.854,Z 450.715,A -85,B 0,C 180,E1 16531.941,E2 16531.941} C_VEL
LIN {X 0,Y 355.29,Z 455.032,A -85,B 0,C 180,E1 16530.774,E2 16530.774} C_VEL
LIN {X 0,Y 365.866,Z 469.466,A -85,B 0,C 180,E1 16527.983,E2 16527.983} C_VEL
LIN {X 0,Y 377.202,Z 486.022,A -85,B 0,C 180,E1 16525.257,E2 16525.257} C_VEL
LIN {X 0,Y 388.874,Z 504.446,A -85,B 0,C 180,E1 16522.689,E2 16522.689} C_VEL
LIN {X 0,Y 394.512,Z 514.358,A -85,B 0,C 180,E1 16521.508,E2 16521.508} C_VEL
LIN {X 0,Y 384.512,Z 741.648,A -85,B 0,C 180,E1 16517.082,E2 16517.082} C_VEL
LIN {X 0,Y 382.953,Z 764.014,A -85,B 0,C 180,E1 16516.548,E2 16516.548} C_VEL
LIN {X 0,Y 380.402,Z 786.106,A -85,B 0,C 180,E1 16515.795,E2 16515.795} C_VEL
LIN {X 0,Y 377.334,Z 807.081,A -85,B 0,C 180,E1 16514.82,E2 16514.82} C_VEL
LIN {X 0,Y 373.637,Z 828,A -85,B 0,C 180,E1 16513.56,E2 16513.56} C_VEL
LIN {X 0,Y 369.704,Z 846.972,A -85,B 0,C 180,E1 16512.125,E2 16512.125} C_VEL
LIN {X 0,Y 365.064,Z 867.108,A -85,B 0,C 180,E1 16510.271,E2 16510.271} C_VEL
LIN {X 0,Y 360.702,Z 884.868,A -85,B 0,C 180,E1 16508.295,E2 16508.295} C_VEL
LIN {X 0,Y 356.213,Z 901.843,A -85,B 0,C 180,E1 16506.022,E2 16506.022} C_VEL
LIN {X 0,Y 351.851,Z 917.962,A -85,B 0,C 180,E1 16503.459,E2 16503.459} C_VEL
LIN {X 0,Y 347.777,Z 933.159,A -85,B 0,C 180,E1 16500.592,E2 16500.592} C_VEL
LIN {X 0,Y 344.232,Z 946.889,A -85,B 0,C 180,E1 16497.508,E2 16497.508} C_VEL
LIN {X 0,Y 341.291,Z 959.037,A -85,B 0,C 180,E1 16494.217,E2 16494.217} C_VEL
LIN {X 0,Y 339.035,Z 969.755,A -85,B 0,C 180,E1 16490.729,E2 16490.729} C_VEL
LIN {X 0,Y 337.539,Z 978.584,A -85,B 0,C 180,E1 16487.234,E2 16487.234} C_VEL
LIN {X 0,Y 336.66,Z 985.558,A -85,B 0,C 180,E1 16483.748,E2 16483.748} C_VEL
LIN {X 0,Y 336.245,Z 991.113,A -85,B 0,C 180,E1 16480.108,E2 16480.108} C_VEL
LIN {X 0,Y 336.174,Z 994.693,A -85,B 0,C 180,E1 16476.836,E2 16476.836} C_VEL
LIN {X 0,Y 336.22,Z 996.875,A -85,B 0,C 180,E1 16473.413,E2 16473.413} C_VEL
LIN {X 0,Y 336.251,Z 997.632,A -85,B 0,C 180,E1 16470.174,E2 16470.174} C_VEL
LIN {X 0,Y 336.226,Z 996.86,A -85,B 0,C 180,E1 16466.765,E2 16466.765} C_VEL
LIN {X 0,Y 336.19,Z 994.686,A -85,B 0,C 180,E1 16463.343,E2 16463.343} C_VEL
LIN {X 0,Y 336.258,Z 990.851,A -85,B 0,C 180,E1 16459.9,E2 16459.9} C_VEL
LIN {X 0,Y 336.634,Z 985.548,A -85,B 0,C 180,E1 16456.434,E2 16456.434} C_VEL
LIN {X 0,Y 337.473,Z 978.53,A -85,B 0,C 180,E1 16452.948,E2 16452.948} C_VEL
LIN {X 0,Y 338.917,Z 969.749,A -85,B 0,C 180,E1 16449.452,E2 16449.452} C_VEL
LIN {X 0,Y 340.986,Z 959.727,A -85,B 0,C 180,E1 16446.135,E2 16446.135} C_VEL
LIN {X 0,Y 343.818,Z 947.682,A -85,B 0,C 180,E1 16442.839,E2 16442.839} C_VEL
LIN {X 0,Y 347.288,Z 934.172,A -85,B 0,C 180,E1 16439.735,E2 16439.735} C_VEL
LIN {X 0,Y 351.446,Z 918.826,A -85,B 0,C 180,E1 16436.764,E2 16436.764} C_VEL
LIN {X 0,Y 355.908,Z 902.59,A -85,B 0,C 180,E1 16434.118,E2 16434.118} C_VEL
LIN {X 0,Y 360.477,Z 885.482,A -85,B 0,C 180,E1 16431.796,E2 16431.796} C_VEL
LIN {X 0,Y 365.204,Z 866.885,A -85,B 0,C 180,E1 16429.678,E2 16429.678} C_VEL
LIN {X 0,Y 369.755,Z 847.922,A -85,B 0,C 180,E1 16427.891,E2 16427.891} C_VEL
LIN {X 0,Y 373.943,Z 828.474,A -85,B 0,C 180,E1 16426.388,E2 16426.388} C_VEL
LIN {X 0,Y 377.708,Z 808.325,A -85,B 0,C 180,E1 16425.139,E2 16425.139} C_VEL
LIN {X 0,Y 381.095,Z 786.846,A -85,B 0,C 180,E1 16424.098,E2 16424.098} C_VEL
LIN {X 0,Y 383.838,Z 765.042,A -85,B 0,C 180,E1 16423.323,E2 16423.323} C_VEL
LIN {X 0,Y 385.564,Z 742.448,A -85,B 0,C 180,E1 16422.766,E2 16422.766} C_VEL
LIN {X 0,Y 395.81,Z 528.007,A -85,B 0,C 180,E1 16418.514,E2 16418.514} C_VEL
LIN {X 0,Y 396.453,Z 513.893,A -85,B 0,C 180,E1 16418.212,E2 16418.212} C_VEL
LIN {X 0,Y 388.605,Z 499.94,A -85,B 0,C 180,E1 16416.26,E2 16416.26} C_VEL
LIN {X 0,Y 380.155,Z 486.305,A -85,B 0,C 180,E1 16413.934,E2 16413.934} C_VEL
LIN {X 0,Y 372.383,Z 474.967,A -85,B 0,C 180,E1 16411.527,E2 16411.527} C_VEL
LIN {X 0,Y 366.008,Z 466.391,A -85,B 0,C 180,E1 16409.274,E2 16409.274} C_VEL
LIN {X 0,Y 362.17,Z 461.304,A -85,B 0,C 180,E1 16407.722,E2 16407.722} C_VEL
LIN {X 0,Y 358.072,Z 456.282,A -85,B 0,C 180,E1 16405.912,E2 16405.912} C_VEL
LIN {X 0,Y 355.923,Z 453.158,A -85,B 0,C 180,E1 16404.567,E2 16404.567} C_VEL
LIN {X 0,Y 354.927,Z 451.267,A -85,B 0,C 180,E1 16403.579,E2 16403.579} C_VEL
LIN {X 0,Y 352.761,Z 447.313,A -85,B 0,C 180,E1 16401.098,E2 16401.098} C_VEL
LIN {X 0,Y 351.111,Z 445.207,A -85,B 0,C 180,E1 16399.116,E2 16399.116} C_VEL
LIN {X 0,Y 349.339,Z 441.373,A -85,B 0,C 180,E1 16394.757,E2 16394.757} C_VEL
LIN {X 0,Y 348.63,Z 440.739,A -85,B 0,C 180,E1 16390.409,E2 16390.409} C_VEL
LIN {X 0,Y 349.382,Z 441.622,A -85,B 0,C 180,E1 16386.903,E2 16386.903} C_VEL
LIN {X 0,Y 352.257,Z 446.831,A -85,B 0,C 180,E1 16381.301,E2 16381.301} C_VEL
LIN {X 0,Y 354.457,Z 451.045,A -85,B 0,C 180,E1 16378.545,E2 16378.545} C_VEL
LIN {X 0,Y 356.216,Z 454.534,A -85,B 0,C 180,E1 16376.862,E2 16376.862} C_VEL
LIN {X 0,Y 358.868,Z 457.753,A -85,B 0,C 180,E1 16375.565,E2 16375.565} C_VEL
LIN {X 0,Y 362.606,Z 462.429,A -85,B 0,C 180,E1 16373.905,E2 16373.905} C_VEL
LIN {X 0,Y 367.462,Z 468.996,A -85,B 0,C 180,E1 16371.987,E2 16371.987} C_VEL
LIN {X 0,Y 375.186,Z 479.734,A -85,B 0,C 180,E1 16369.326,E2 16369.326} C_VEL
LIN {X 0,Y 383.637,Z 492.918,A -85,B 0,C 180,E1 16366.779,E2 16366.779} C_VEL
LIN {X 0,Y 391.727,Z 506.535,A -85,B 0,C 180,E1 16364.606,E2 16364.606} C_VEL
LIN {X 0,Y 394.819,Z 512.547,A -85,B 0,C 180,E1 16363.812,E2 16363.812} C_VEL
LIN {X 0,Y 382.57,Z 726.111,A -85,B 0,C 180,E1 16359.352,E2 16359.352} C_VEL
LIN {X 0,Y 380.544,Z 746.844,A -85,B 0,C 180,E1 16358.662,E2 16358.662} C_VEL
LIN {X 0,Y 377.857,Z 766.948,A -85,B 0,C 180,E1 16357.738,E2 16357.738} C_VEL
LIN {X 0,Y 374.484,Z 787.202,A -85,B 0,C 180,E1 16356.517,E2 16356.517} C_VEL
LIN {X 0,Y 370.725,Z 806.184,A -85,B 0,C 180,E1 16355.074,E2 16355.074} C_VEL
LIN {X 0,Y 366.692,Z 823.946,A -85,B 0,C 180,E1 16353.415,E2 16353.415} C_VEL
LIN {X 0,Y 362.181,Z 841.711,A -85,B 0,C 180,E1 16351.378,E2 16351.378} C_VEL
LIN {X 0,Y 357.87,Z 857.305,A -85,B 0,C 180,E1 16349.209,E2 16349.209} C_VEL
LIN {X 0,Y 353.54,Z 872.187,A -85,B 0,C 180,E1 16346.724,E2 16346.724} C_VEL
LIN {X 0,Y 349.324,Z 886.296,A -85,B 0,C 180,E1 16343.869,E2 16343.869} C_VEL
LIN {X 0,Y 345.628,Z 898.647,A -85,B 0,C 180,E1 16340.824,E2 16340.824} C_VEL
LIN {X 0,Y 342.737,Z 908.692,A -85,B 0,C 180,E1 16337.808,E2 16337.808} C_VEL
LIN {X 0,Y 340.289,Z 917.77,A -85,B 0,C 180,E1 16334.438,E2 16334.438} C_VEL
LIN {X 0,Y 338.488,Z 925.242,A -85,B 0,C 180,E1 16330.869,E2 16330.869} C_VEL
LIN {X 0,Y 337.389,Z 930.633,A -85,B 0,C 180,E1 16327.404,E2 16327.404} C_VEL
LIN {X 0,Y 336.792,Z 934.398,A -85,B 0,C 180,E1 16323.921,E2 16323.921} C_VEL
LIN {X 0,Y 336.502,Z 936.634,A -85,B 0,C 180,E1 16320.334,E2 16320.334} C_VEL
LIN {X 0,Y 336.43,Z 937.273,A -85,B 0,C 180,E1 16317.041,E2 16317.041} C_VEL
LIN {X 0,Y 336.471,Z 936.381,A -85,B 0,C 180,E1 16313.646,E2 16313.646} C_VEL
LIN {X 0,Y 336.716,Z 933.941,A -85,B 0,C 180,E1 16310.144,E2 16310.144} C_VEL
LIN {X 0,Y 337.237,Z 929.994,A -85,B 0,C 180,E1 16306.709,E2 16306.709} C_VEL
LIN {X 0,Y 338.205,Z 924.517,A -85,B 0,C 180,E1 16303.328,E2 16303.328} C_VEL
LIN {X 0,Y 339.814,Z 916.926,A -85,B 0,C 180,E1 16299.822,E2 16299.822} C_VEL
LIN {X 0,Y 342.001,Z 907.899,A -85,B 0,C 180,E1 16296.543,E2 16296.543} C_VEL
LIN {X 0,Y 344.721,Z 897.557,A -85,B 0,C 180,E1 16293.488,E2 16293.488} C_VEL
LIN {X 0,Y 348.108,Z 885.219,A -85,B 0,C 180,E1 16290.49,E2 16290.49} C_VEL
LIN {X 0,Y 351.694,Z 872.291,A -85,B 0,C 180,E1 16287.879,E2 16287.879} C_VEL
LIN {X 0,Y 355.807,Z 857.069,A -85,B 0,C 180,E1 16285.322,E2 16285.322} C_VEL
LIN {X 0,Y 359.995,Z 840.708,A -85,B 0,C 180,E1 16283.058,E2 16283.058} C_VEL
LIN {X 0,Y 360.199,Z 839.917,A -85,B 0,C 180,E1 16282.955,E2 16282.955} C_VEL
LIN {X 0,Y 360.815,Z 834.077,A -85,B 0,C 180,E1 16282.146,E2 16282.146} C_VEL
LIN {X 0,Y 359.508,Z 819.412,A -85,B 0,C 180,E1 16279.967,E2 16279.967} C_VEL
LIN {X 0,Y 360.075,Z 813.133,A -85,B 0,C 180,E1 16279.252,E2 16279.252} C_VEL
LIN {X 0,Y 363.822,Z 794.914,A -85,B 0,C 180,E1 16277.721,E2 16277.721} C_VEL
LIN {X 0,Y 367.325,Z 775.032,A -85,B 0,C 180,E1 16276.379,E2 16276.379} C_VEL
LIN {X 0,Y 370.226,Z 754.79,A -85,B 0,C 180,E1 16275.316,E2 16275.316} C_VEL
LIN {X 0,Y 372.526,Z 733.911,A -85,B 0,C 180,E1 16274.505,E2 16274.505} C_VEL
LIN {X 0,Y 374.117,Z 711.861,A -85,B 0,C 180,E1 16273.929,E2 16273.929} C_VEL
LIN {X 0,Y 384.126,Z 512.465,A -85,B 0,C 180,E1 16269.877,E2 16269.877} C_VEL
LIN {X 0,Y 372.855,Z 493.339,A -85,B 0,C 180,E1 16267.342,E2 16267.342} C_VEL
LIN {X 0,Y 361.667,Z 476.193,A -85,B 0,C 180,E1 16264.609,E2 16264.609} C_VEL
LIN {X 0,Y 352.057,Z 462.598,A -85,B 0,C 180,E1 16262.039,E2 16262.039} C_VEL
LIN {X 0,Y 344.884,Z 452.698,A -85,B 0,C 180,E1 16259.895,E2 16259.895} C_VEL
LIN {X 0,Y 340.511,Z 444.113,A -85,B 0,C 180,E1 16257.094,E2 16257.094} C_VEL
LIN {X 0,Y 337.9,Z 439.255,A -85,B 0,C 180,E1 16255.348,E2 16255.348} C_VEL
LIN {X 0,Y 335.426,Z 434.621,A -85,B 0,C 180,E1 16253.595,E2 16253.595} C_VEL
LIN {X 0,Y 333.304,Z 431.034,A -85,B 0,C 180,E1 16252.089,E2 16252.089} C_VEL
LIN {X 0,Y 332.465,Z 429.435,A -85,B 0,C 180,E1 16251.438,E2 16251.438} C_VEL
LIN {X 0,Y 330.355,Z 426.002,A -85,B 0,C 180,E1 16249.856,E2 16249.856} C_VEL
LIN {X 0,Y 330.064,Z 424.775,A -85,B 0,C 180,E1 16249.229,E2 16249.229} C_VEL
LIN {X 0,Y 330.043,Z 424.609,A -85,B 0,C 180,E1 16244.851,E2 16244.851} C_VEL
LIN {X 0,Y 330.052,Z 424.6,A -85,B 0,C 180,E1 16240.413,E2 16240.413} C_VEL
LIN {X 0,Y 330.045,Z 424.592,A -85,B 0,C 180,E1 16235.996,E2 16235.996} C_VEL
LIN {X 0,Y 330.046,Z 424.589,A -85,B 0,C 180,E1 16231.608,E2 16231.608} C_VEL
LIN {X 0,Y 330.048,Z 424.599,A -85,B 0,C 180,E1 16227.223,E2 16227.223} C_VEL
LIN {X 0,Y 330.056,Z 424.621,A -85,B 0,C 180,E1 16222.816,E2 16222.816} C_VEL
LIN {X 0,Y 330.046,Z 424.605,A -85,B 0,C 180,E1 16218.365,E2 16218.365} C_VEL
LIN {X 0,Y 330.044,Z 424.588,A -85,B 0,C 180,E1 16214.026,E2 16214.026} C_VEL
LIN {X 0,Y 330.044,Z 424.593,A -85,B 0,C 180,E1 16209.768,E2 16209.768} C_VEL
LIN {X 0,Y 330.047,Z 424.615,A -85,B 0,C 180,E1 16205.389,E2 16205.389} C_VEL
LIN {X 0,Y 330.052,Z 424.614,A -85,B 0,C 180,E1 16201.042,E2 16201.042} C_VEL
LIN {X 0,Y 330.042,Z 424.597,A -85,B 0,C 180,E1 16196.701,E2 16196.701} C_VEL
LIN {X 0,Y 330.041,Z 424.592,A -85,B 0,C 180,E1 16192.34,E2 16192.34} C_VEL
LIN {X 0,Y 330.04,Z 424.594,A -85,B 0,C 180,E1 16187.935,E2 16187.935} C_VEL
LIN {X 0,Y 330.072,Z 424.83,A -85,B 0,C 180,E1 16183.8,E2 16183.8} C_VEL
LIN {X 0,Y 331.645,Z 428.493,A -85,B 0,C 180,E1 16182.272,E2 16182.272} C_VEL
LIN {X 0,Y 333.252,Z 430.479,A -85,B 0,C 180,E1 16181.275,E2 16181.275} C_VEL
LIN {X 0,Y 335.314,Z 434.373,A -85,B 0,C 180,E1 16179.764,E2 16179.764} C_VEL
LIN {X 0,Y 336.39,Z 435.893,A -85,B 0,C 180,E1 16179.104,E2 16179.104} C_VEL
LIN {X 0,Y 338.654,Z 439.928,A -85,B 0,C 180,E1 16177.613,E2 16177.613} C_VEL
LIN {X 0,Y 342.344,Z 446.665,A -85,B 0,C 180,E1 16175.314,E2 16175.314} C_VEL
LIN {X 0,Y 347.09,Z 454.882,A -85,B 0,C 180,E1 16172.74,E2 16172.74} C_VEL
LIN {X 0,Y 358.652,Z 470.677,A -85,B 0,C 180,E1 16169.464,E2 16169.464} C_VEL
LIN {X 0,Y 369.467,Z 486.128,A -85,B 0,C 180,E1 16166.724,E2 16166.724} C_VEL
LIN {X 0,Y 380.979,Z 504.165,A -85,B 0,C 180,E1 16164.041,E2 16164.041} C_VEL
LIN {X 0,Y 388.949,Z 517.654,A -85,B 0,C 180,E1 16162.308,E2 16162.308} C_VEL
LIN {X 0,Y 378.16,Z 750.377,A -85,B 0,C 180,E1 16157.712,E2 16157.712} C_VEL
LIN {X 0,Y 376.096,Z 772.811,A -85,B 0,C 180,E1 16157.088,E2 16157.088} C_VEL
LIN {X 0,Y 373.306,Z 793.995,A -85,B 0,C 180,E1 16156.264,E2 16156.264} C_VEL
LIN {X 0,Y 370.038,Z 813.813,A -85,B 0,C 180,E1 16155.235,E2 16155.235} C_VEL
LIN {X 0,Y 366.127,Z 833.76,A -85,B 0,C 180,E1 16153.923,E2 16153.923} C_VEL
LIN {X 0,Y 361.727,Z 853.615,A -85,B 0,C 180,E1 16152.307,E2 16152.307} C_VEL
LIN {X 0,Y 357.05,Z 872.643,A -85,B 0,C 180,E1 16150.415,E2 16150.415} C_VEL
LIN {X 0,Y 352.425,Z 890.062,A -85,B 0,C 180,E1 16148.312,E2 16148.312} C_VEL
LIN {X 0,Y 347.469,Z 907.86,A -85,B 0,C 180,E1 16145.745,E2 16145.745} C_VEL
LIN {X 0,Y 343.299,Z 922.698,A -85,B 0,C 180,E1 16143.202,E2 16143.202} C_VEL
LIN {X 0,Y 339.24,Z 937.041,A -85,B 0,C 180,E1 16140.268,E2 16140.268} C_VEL
LIN {X 0,Y 335.68,Z 950.242,A -85,B 0,C 180,E1 16137.052,E2 16137.052} C_VEL
LIN {X 0,Y 332.777,Z 962.092,A -85,B 0,C 180,E1 16133.596,E2 16133.596} C_VEL
LIN {X 0,Y 330.633,Z 972.315,A -85,B 0,C 180,E1 16129.985,E2 16129.985} C_VEL
LIN {X 0,Y 329.251,Z 980.558,A -85,B 0,C 180,E1 16126.34,E2 16126.34} C_VEL
LIN {X 0,Y 328.488,Z 987.127,A -85,B 0,C 180,E1 16122.663,E2 16122.663} C_VEL
LIN {X 0,Y 328.223,Z 991.734,A -85,B 0,C 180,E1 16119.254,E2 16119.254} C_VEL
LIN {X 0,Y 328.209,Z 994.879,A -85,B 0,C 180,E1 16115.773,E2 16115.773} C_VEL
LIN {X 0,Y 328.251,Z 996.574,A -85,B 0,C 180,E1 16112.448,E2 16112.448} C_VEL
LIN {X 0,Y 328.278,Z 996.816,A -85,B 0,C 180,E1 16109.131,E2 16109.131} C_VEL
LIN {X 0,Y 328.243,Z 995.833,A -85,B 0,C 180,E1 16105.986,E2 16105.986} C_VEL
LIN {X 0,Y 328.194,Z 993.276,A -85,B 0,C 180,E1 16102.477,E2 16102.477} C_VEL
LIN {X 0,Y 328.33,Z 989.441,A -85,B 0,C 180,E1 16099.121,E2 16099.121} C_VEL
LIN {X 0,Y 328.82,Z 983.495,A -85,B 0,C 180,E1 16095.386,E2 16095.386} C_VEL
LIN {X 0,Y 329.837,Z 976.197,A -85,B 0,C 180,E1 16091.811,E2 16091.811} C_VEL
LIN {X 0,Y 331.559,Z 967.034,A -85,B 0,C 180,E1 16088.232,E2 16088.232} C_VEL
LIN {X 0,Y 334.079,Z 955.929,A -85,B 0,C 180,E1 16084.668,E2 16084.668} C_VEL
LIN {X 0,Y 337.327,Z 943.383,A -85,B 0,C 180,E1 16081.308,E2 16081.308} C_VEL
LIN {X 0,Y 341.242,Z 929.426,A -85,B 0,C 180,E1 16078.175,E2 16078.175} C_VEL
LIN {X 0,Y 345.687,Z 913.871,A -85,B 0,C 180,E1 16075.269,E2 16075.269} C_VEL
LIN {X 0,Y 350.406,Z 897.4,A -85,B 0,C 180,E1 16072.679,E2 16072.679} C_VEL
LIN {X 0,Y 355.232,Z 880.142,A -85,B 0,C 180,E1 16070.399,E2 16070.399} C_VEL
LIN {X 0,Y 360.198,Z 861.38,A -85,B 0,C 180,E1 16068.338,E2 16068.338} C_VEL
LIN {X 0,Y 364.746,Z 842.54,A -85,B 0,C 180,E1 16066.638,E2 16066.638} C_VEL
LIN {X 0,Y 369.173,Z 822.118,A -85,B 0,C 180,E1 16065.134,E2 16065.134} C_VEL
LIN {X 0,Y 373.037,Z 801.611,A -85,B 0,C 180,E1 16063.93,E2 16063.93} C_VEL
LIN {X 0,Y 376.302,Z 780.427,A -85,B 0,C 180,E1 16062.988,E2 16062.988} C_VEL
LIN {X 0,Y 378.877,Z 758.459,A -85,B 0,C 180,E1 16062.279,E2 16062.279} C_VEL
LIN {X 0,Y 380.532,Z 733.32,A -85,B 0,C 180,E1 16061.705,E2 16061.705} C_VEL
LIN {X 0,Y 390.932,Z 526.731,A -85,B 0,C 180,E1 16057.568,E2 16057.568} C_VEL
LIN {X 0,Y 391.289,Z 517.346,A -85,B 0,C 180,E1 16057.348,E2 16057.348} C_VEL
LIN {X 0,Y 382.851,Z 502.329,A -85,B 0,C 180,E1 16055.114,E2 16055.114} C_VEL
LIN {X 0,Y 375.368,Z 490.394,A -85,B 0,C 180,E1 16052.914,E2 16052.914} C_VEL
LIN {X 0,Y 368.77,Z 480.578,A -85,B 0,C 180,E1 16050.736,E2 16050.736} C_VEL
LIN {X 0,Y 363.474,Z 473.325,A -85,B 0,C 180,E1 16048.776,E2 16048.776} C_VEL
LIN {X 0,Y 359.8,Z 468.363,A -85,B 0,C 180,E1 16047.231,E2 16047.231} C_VEL
LIN {X 0,Y 356.119,Z 463.673,A -85,B 0,C 180,E1 16045.529,E2 16045.529} C_VEL
LIN {X 0,Y 352.205,Z 458.724,A -85,B 0,C 180,E1 16043.418,E2 16043.418} C_VEL
LIN {X 0,Y 348.802,Z 454.588,A -85,B 0,C 180,E1 16041.173,E2 16041.173} C_VEL
LIN {X 0,Y 348.08,Z 453.253,A -85,B 0,C 180,E1 16040.338,E2 16040.338} C_VEL
LIN {X 0,Y 345.308,Z 448.284,A -85,B 0,C 180,E1 16034.755,E2 16034.755} C_VEL
LIN {X 0,Y 344.587,Z 447.643,A -85,B 0,C 180,E1 16030.363,E2 16030.363} C_VEL
LIN {X 0,Y 345.262,Z 448.472,A -85,B 0,C 180,E1 16026.986,E2 16026.986} C_VEL
LIN {X 0,Y 347.968,Z 453.634,A -85,B 0,C 180,E1 16021.399,E2 16021.399} C_VEL
LIN {X 0,Y 351.652,Z 458.409,A -85,B 0,C 180,E1 16018.778,E2 16018.778} C_VEL
LIN {X 0,Y 356.673,Z 464.9,A -85,B 0,C 180,E1 16016.021,E2 16016.021} C_VEL
LIN {X 0,Y 360.411,Z 469.731,A -85,B 0,C 180,E1 16014.308,E2 16014.308} C_VEL
LIN {X 0,Y 365.05,Z 476.164,A -85,B 0,C 180,E1 16012.402,E2 16012.402} C_VEL
LIN {X 0,Y 372.244,Z 486.43,A -85,B 0,C 180,E1 16009.827,E2 16009.827} C_VEL
LIN {X 0,Y 380.363,Z 499.404,A -85,B 0,C 180,E1 16007.285,E2 16007.285} C_VEL
LIN {X 0,Y 388.233,Z 512.998,A -85,B 0,C 180,E1 16005.094,E2 16005.094} C_VEL
LIN {X 0,Y 389.778,Z 516.308,A -85,B 0,C 180,E1 16004.672,E2 16004.672} C_VEL
LIN {X 0,Y 377.134,Z 726.522,A -85,B 0,C 180,E1 16000.236,E2 16000.236} C_VEL
LIN {X 0,Y 375.005,Z 747.439,A -85,B 0,C 180,E1 15999.533,E2 15999.533} C_VEL
LIN {X 0,Y 372.262,Z 767.222,A -85,B 0,C 180,E1 15998.619,E2 15998.619} C_VEL
LIN {X 0,Y 368.757,Z 787.512,A -85,B 0,C 180,E1 15997.392,E2 15997.392} C_VEL
LIN {X 0,Y 364.987,Z 805.841,A -85,B 0,C 180,E1 15995.995,E2 15995.995} C_VEL
LIN {X 0,Y 360.659,Z 824.132,A -85,B 0,C 180,E1 15994.278,E2 15994.278} C_VEL
LIN {X 0,Y 355.936,Z 841.926,A -85,B 0,C 180,E1 15992.224,E2 15992.224} C_VEL
LIN {X 0,Y 351.394,Z 857.635,A -85,B 0,C 180,E1 15990.019,E2 15990.019} C_VEL
LIN {X 0,Y 346.842,Z 872.487,A -85,B 0,C 180,E1 15987.512,E2 15987.512} C_VEL
LIN {X 0,Y 342.496,Z 886.326,A -85,B 0,C 180,E1 15984.688,E2 15984.688} C_VEL
LIN {X 0,Y 338.712,Z 898.277,A -85,B 0,C 180,E1 15981.733,E2 15981.733} C_VEL
LIN {X 0,Y 335.488,Z 908.76,A -85,B 0,C 180,E1 15978.575,E2 15978.575} C_VEL
LIN {X 0,Y 332.772,Z 918.057,A -85,B 0,C 180,E1 15975.082,E2 15975.082} C_VEL
LIN {X 0,Y 330.89,Z 925.187,A -85,B 0,C 180,E1 15971.659,E2 15971.659} C_VEL
LIN {X 0,Y 329.655,Z 930.654,A -85,B 0,C 180,E1 15968.218,E2 15968.218} C_VEL
LIN {X 0,Y 328.924,Z 934.7,A -85,B 0,C 180,E1 15964.636,E2 15964.636} C_VEL
LIN {X 0,Y 328.596,Z 937.11,A -85,B 0,C 180,E1 15961.144,E2 15961.144} C_VEL
LIN {X 0,Y 328.465,Z 937.934,A -85,B 0,C 180,E1 15957.753,E2 15957.753} C_VEL
LIN {X 0,Y 328.49,Z 937.368,A -85,B 0,C 180,E1 15954.257,E2 15954.257} C_VEL
LIN {X 0,Y 328.679,Z 935.421,A -85,B 0,C 180,E1 15950.845,E2 15950.845} C_VEL
LIN {X 0,Y 329.17,Z 931.792,A -85,B 0,C 180,E1 15947.314,E2 15947.314} C_VEL
LIN {X 0,Y 330.072,Z 926.623,A -85,B 0,C 180,E1 15943.841,E2 15943.841} C_VEL
LIN {X 0,Y 331.639,Z 919.47,A -85,B 0,C 180,E1 15940.242,E2 15940.242} C_VEL
LIN {X 0,Y 333.801,Z 910.919,A -85,B 0,C 180,E1 15936.878,E2 15936.878} C_VEL
LIN {X 0,Y 336.63,Z 900.671,A -85,B 0,C 180,E1 15933.627,E2 15933.627} C_VEL
LIN {X 0,Y 340.117,Z 888.574,A -85,B 0,C 180,E1 15930.502,E2 15930.502} C_VEL
LIN {X 0,Y 343.989,Z 875.167,A -85,B 0,C 180,E1 15927.664,E2 15927.664} C_VEL
LIN {X 0,Y 348.056,Z 860.78,A -85,B 0,C 180,E1 15925.135,E2 15925.135} C_VEL
LIN {X 0,Y 352.349,Z 844.98,A -85,B 0,C 180,E1 15922.824,E2 15922.824} C_VEL
LIN {X 0,Y 356.708,Z 827.63,A -85,B 0,C 180,E1 15920.722,E2 15920.722} C_VEL
LIN {X 0,Y 360.075,Z 813.133,A -85,B 0,C 180,E1 15919.252,E2 15919.252} C_VEL
LIN {X 0,Y 360.732,Z 806.72,A -85,B 0,C 180,E1 15918.563,E2 15918.563} C_VEL
LIN {X 0,Y 359.398,Z 790.604,A -85,B 0,C 180,E1 15916.659,E2 15916.659} C_VEL
LIN {X 0,Y 359.844,Z 783.79,A -85,B 0,C 180,E1 15916.078,E2 15916.078} C_VEL
LIN {X 0,Y 363.069,Z 764.033,A -85,B 0,C 180,E1 15914.912,E2 15914.912} C_VEL
LIN {X 0,Y 365.786,Z 742.956,A -85,B 0,C 180,E1 15913.971,E2 15913.971} C_VEL
LIN {X 0,Y 367.684,Z 722.383,A -85,B 0,C 180,E1 15913.315,E2 15913.315} C_VEL
LIN {X 0,Y 378.619,Z 515.957,A -85,B 0,C 180,E1 15909.051,E2 15909.051} C_VEL
LIN {X 0,Y 367.856,Z 497.702,A -85,B 0,C 180,E1 15906.543,E2 15906.543} C_VEL
LIN {X 0,Y 357.842,Z 482.18,A -85,B 0,C 180,E1 15904.012,E2 15904.012} C_VEL
LIN {X 0,Y 348.71,Z 469.09,A -85,B 0,C 180,E1 15901.503,E2 15901.503} C_VEL
LIN {X 0,Y 341.068,Z 458.696,A -85,B 0,C 180,E1 15899.199,E2 15899.199} C_VEL
LIN {X 0,Y 336.557,Z 452.579,A -85,B 0,C 180,E1 15897.67,E2 15897.67} C_VEL
LIN {X 0,Y 332.841,Z 445.3,A -85,B 0,C 180,E1 15895.095,E2 15895.095} C_VEL
LIN {X 0,Y 330.087,Z 440.35,A -85,B 0,C 180,E1 15893.144,E2 15893.144} C_VEL
LIN {X 0,Y 327.473,Z 435.549,A -85,B 0,C 180,E1 15891.132,E2 15891.132} C_VEL
LIN {X 0,Y 325.327,Z 431.679,A -85,B 0,C 180,E1 15889.388,E2 15889.388} C_VEL
LIN {X 0,Y 322.397,Z 426.956,A -85,B 0,C 180,E1 15886.974,E2 15886.974} C_VEL
LIN {X 0,Y 322.135,Z 425.776,A -85,B 0,C 180,E1 15886.32,E2 15886.32} C_VEL
LIN {X 0,Y 322.11,Z 425.578,A -85,B 0,C 180,E1 15881.839,E2 15881.839} C_VEL
LIN {X 0,Y 322.107,Z 425.582,A -85,B 0,C 180,E1 15877.475,E2 15877.475} C_VEL
LIN {X 0,Y 322.109,Z 425.596,A -85,B 0,C 180,E1 15873.055,E2 15873.055} C_VEL
LIN {X 0,Y 322.111,Z 425.612,A -85,B 0,C 180,E1 15868.539,E2 15868.539} C_VEL
LIN {X 0,Y 322.107,Z 425.589,A -85,B 0,C 180,E1 15864.126,E2 15864.126} C_VEL
LIN {X 0,Y 322.106,Z 425.574,A -85,B 0,C 180,E1 15859.777,E2 15859.777} C_VEL
LIN {X 0,Y 322.111,Z 425.581,A -85,B 0,C 180,E1 15855.483,E2 15855.483} C_VEL
LIN {X 0,Y 322.108,Z 425.607,A -85,B 0,C 180,E1 15851.097,E2 15851.097} C_VEL
LIN {X 0,Y 322.106,Z 425.602,A -85,B 0,C 180,E1 15846.596,E2 15846.596} C_VEL
LIN {X 0,Y 322.104,Z 425.581,A -85,B 0,C 180,E1 15842.135,E2 15842.135} C_VEL
LIN {X 0,Y 322.104,Z 425.576,A -85,B 0,C 180,E1 15837.866,E2 15837.866} C_VEL
LIN {X 0,Y 322.109,Z 425.581,A -85,B 0,C 180,E1 15833.387,E2 15833.387} C_VEL
LIN {X 0,Y 322.108,Z 425.588,A -85,B 0,C 180,E1 15828.904,E2 15828.904} C_VEL
LIN {X 0,Y 322.168,Z 425.965,A -85,B 0,C 180,E1 15826.723,E2 15826.723} C_VEL
LIN {X 0,Y 323.862,Z 429.681,A -85,B 0,C 180,E1 15824.97,E2 15824.97} C_VEL
LIN {X 0,Y 325.404,Z 431.369,A -85,B 0,C 180,E1 15823.947,E2 15823.947} C_VEL
LIN {X 0,Y 327.205,Z 435.122,A -85,B 0,C 180,E1 15822.392,E2 15822.392} C_VEL
LIN {X 0,Y 328.517,Z 436.784,A -85,B 0,C 180,E1 15821.547,E2 15821.547} C_VEL
LIN {X 0,Y 330.578,Z 440.677,A -85,B 0,C 180,E1 15820.015,E2 15820.015} C_VEL
LIN {X 0,Y 331.812,Z 442.76,A -85,B 0,C 180,E1 15819.172,E2 15819.172} C_VEL
LIN {X 0,Y 334.604,Z 447.707,A -85,B 0,C 180,E1 15817.327,E2 15817.327} C_VEL
LIN {X 0,Y 337.541,Z 453.042,A -85,B 0,C 180,E1 15815.5,E2 15815.5} C_VEL
LIN {X 0,Y 339.964,Z 456.407,A -85,B 0,C 180,E1 15814.525,E2 15814.525} C_VEL
LIN {X 0,Y 348.804,Z 468.188,A -85,B 0,C 180,E1 15811.819,E2 15811.819} C_VEL
LIN {X 0,Y 359.123,Z 482.658,A -85,B 0,C 180,E1 15808.952,E2 15808.952} C_VEL
LIN {X 0,Y 369.578,Z 498.289,A -85,B 0,C 180,E1 15806.317,E2 15806.317} C_VEL
LIN {X 0,Y 381.28,Z 517.209,A -85,B 0,C 180,E1 15803.608,E2 15803.608} C_VEL
LIN {X 0,Y 383.432,Z 521.376,A -85,B 0,C 180,E1 15803.122,E2 15803.122} C_VEL
LIN {X 0,Y 372.243,Z 752.091,A -85,B 0,C 180,E1 15798.516,E2 15798.516} C_VEL
LIN {X 0,Y 370.079,Z 773.796,A -85,B 0,C 180,E1 15797.888,E2 15797.888} C_VEL
LIN {X 0,Y 367.031,Z 795.561,A -85,B 0,C 180,E1 15797.01,E2 15797.01} C_VEL
LIN {X 0,Y 363.675,Z 815.133,A -85,B 0,C 180,E1 15795.971,E2 15795.971} C_VEL
LIN {X 0,Y 359.517,Z 835.272,A -85,B 0,C 180,E1 15794.606,E2 15794.606} C_VEL
LIN {X 0,Y 354.723,Z 855.802,A -85,B 0,C 180,E1 15792.874,E2 15792.874} C_VEL
LIN {X 0,Y 349.964,Z 874.242,A -85,B 0,C 180,E1 15790.975,E2 15790.975} C_VEL
LIN {X 0,Y 345.022,Z 892.033,A -85,B 0,C 180,E1 15788.756,E2 15788.756} C_VEL
LIN {X 0,Y 340.231,Z 908.356,A -85,B 0,C 180,E1 15786.314,E2 15786.314} C_VEL
LIN {X 0,Y 335.428,Z 924.551,A -85,B 0,C 180,E1 15783.423,E2 15783.423} C_VEL
LIN {X 0,Y 331.356,Z 938.496,A -85,B 0,C 180,E1 15780.463,E2 15780.463} C_VEL
LIN {X 0,Y 327.768,Z 951.129,A -85,B 0,C 180,E1 15777.234,E2 15777.234} C_VEL
LIN {X 0,Y 324.855,Z 962.441,A -85,B 0,C 180,E1 15773.782,E2 15773.782} C_VEL
LIN {X 0,Y 322.678,Z 972.341,A -85,B 0,C 180,E1 15770.136,E2 15770.136} C_VEL
LIN {X 0,Y 321.274,Z 980.386,A -85,B 0,C 180,E1 15766.455,E2 15766.455} C_VEL
LIN {X 0,Y 320.511,Z 986.644,A -85,B 0,C 180,E1 15762.8,E2 15762.8} C_VEL
LIN {X 0,Y 320.234,Z 991.368,A -85,B 0,C 180,E1 15759.166,E2 15759.166} C_VEL
LIN {X 0,Y 320.232,Z 994.393,A -85,B 0,C 180,E1 15755.558,E2 15755.558} C_VEL
LIN {X 0,Y 320.296,Z 995.99,A -85,B 0,C 180,E1 15751.972,E2 15751.972} C_VEL
LIN {X 0,Y 320.313,Z 996.046,A -85,B 0,C 180,E1 15748.752,E2 15748.752} C_VEL
LIN {X 0,Y 320.245,Z 994.873,A -85,B 0,C 180,E1 15745.348,E2 15745.348} C_VEL
LIN {X 0,Y 320.239,Z 992.024,A -85,B 0,C 180,E1 15741.747,E2 15741.747} C_VEL
LIN {X 0,Y 320.436,Z 987.463,A -85,B 0,C 180,E1 15737.937,E2 15737.937} C_VEL
LIN {X 0,Y 321.065,Z 981.443,A -85,B 0,C 180,E1 15734.285,E2 15734.285} C_VEL
LIN {X 0,Y 322.399,Z 973.283,A -85,B 0,C 180,E1 15730.436,E2 15730.436} C_VEL
LIN {X 0,Y 324.52,Z 963.348,A -85,B 0,C 180,E1 15726.656,E2 15726.656} C_VEL
LIN {X 0,Y 327.435,Z 951.955,A -85,B 0,C 180,E1 15723.081,E2 15723.081} C_VEL
LIN {X 0,Y 331.084,Z 938.937,A -85,B 0,C 180,E1 15719.718,E2 15719.718} C_VEL
LIN {X 0,Y 335.453,Z 924.267,A -85,B 0,C 180,E1 15716.541,E2 15716.541} C_VEL
LIN {X 0,Y 340.22,Z 908.595,A -85,B 0,C 180,E1 15713.694,E2 15713.694} C_VEL
LIN {X 0,Y 345.405,Z 891.456,A -85,B 0,C 180,E1 15711.092,E2 15711.092} C_VEL
LIN {X 0,Y 350.457,Z 873.77,A -85,B 0,C 180,E1 15708.867,E2 15708.867} C_VEL
LIN {X 0,Y 355.537,Z 854.909,A -85,B 0,C 180,E1 15706.898,E2 15706.898} C_VEL
LIN {X 0,Y 360.405,Z 835.142,A -85,B 0,C 180,E1 15705.204,E2 15705.204} C_VEL
LIN {X 0,Y 364.778,Z 815.042,A -85,B 0,C 180,E1 15703.82,E2 15703.82} C_VEL
LIN {X 0,Y 368.374,Z 795.437,A -85,B 0,C 180,E1 15702.755,E2 15702.755} C_VEL
LIN {X 0,Y 371.578,Z 774.436,A -85,B 0,C 180,E1 15701.882,E2 15701.882} C_VEL
LIN {X 0,Y 374.012,Z 752.321,A -85,B 0,C 180,E1 15701.218,E2 15701.218} C_VEL
LIN {X 0,Y 377.481,Z 686.648,A -85,B 0,C 180,E1 15699.864,E2 15699.864} C_VEL
LIN {X 0,Y 386.418,Z 521.227,A -85,B 0,C 180,E1 15696.498,E2 15696.498} C_VEL
LIN {X 0,Y 378.713,Z 507.401,A -85,B 0,C 180,E1 15694.355,E2 15694.355} C_VEL
LIN {X 0,Y 372.116,Z 496.638,A -85,B 0,C 180,E1 15692.323,E2 15692.323} C_VEL
LIN {X 0,Y 365.14,Z 485.97,A -85,B 0,C 180,E1 15689.892,E2 15689.892} C_VEL
LIN {X 0,Y 360.456,Z 479.546,A -85,B 0,C 180,E1 15688.045,E2 15688.045} C_VEL
LIN {X 0,Y 357.517,Z 475.483,A -85,B 0,C 180,E1 15686.76,E2 15686.76} C_VEL
LIN {X 0,Y 353.88,Z 470.72,A -85,B 0,C 180,E1 15684.986,E2 15684.986} C_VEL
LIN {X 0,Y 350.357,Z 466.168,A -85,B 0,C 180,E1 15683.015,E2 15683.015} C_VEL
LIN {X 0,Y 346.892,Z 461.62,A -85,B 0,C 180,E1 15680.587,E2 15680.587} C_VEL
LIN {X 0,Y 341.834,Z 455.523,A -85,B 0,C 180,E1 15674.915,E2 15674.915} C_VEL
LIN {X 0,Y 340.778,Z 454.644,A -85,B 0,C 180,E1 15671.165,E2 15671.165} C_VEL
LIN {X 0,Y 341.55,Z 455.291,A -85,B 0,C 180,E1 15667.569,E2 15667.569} C_VEL
LIN {X 0,Y 346.327,Z 461.191,A -85,B 0,C 180,E1 15661.737,E2 15661.737} C_VEL
LIN {X 0,Y 351.051,Z 467.467,A -85,B 0,C 180,E1 15658.424,E2 15658.424} C_VEL
LIN {X 0,Y 354.905,Z 472.644,A -85,B 0,C 180,E1 15656.284,E2 15656.284} C_VEL
LIN {X 0,Y 358.236,Z 477.024,A -85,B 0,C 180,E1 15654.715,E2 15654.715} C_VEL
LIN {X 0,Y 362.806,Z 483.539,A -85,B 0,C 180,E1 15652.764,E2 15652.764} C_VEL
LIN {X 0,Y 369.458,Z 493.318,A -85,B 0,C 180,E1 15650.301,E2 15650.301} C_VEL
LIN {X 0,Y 377.055,Z 505.74,A -85,B 0,C 180,E1 15647.829,E2 15647.829} C_VEL
LIN {X 0,Y 384.524,Z 518.986,A -85,B 0,C 180,E1 15645.66,E2 15645.66} C_VEL
LIN {X 0,Y 384.829,Z 520.198,A -85,B 0,C 180,E1 15645.553,E2 15645.553} C_VEL
LIN {X 0,Y 371.809,Z 727.161,A -85,B 0,C 180,E1 15641.144,E2 15641.144} C_VEL
LIN {X 0,Y 369.603,Z 747.971,A -85,B 0,C 180,E1 15640.439,E2 15640.439} C_VEL
LIN {X 0,Y 366.661,Z 768.265,A -85,B 0,C 180,E1 15639.49,E2 15639.49} C_VEL
LIN {X 0,Y 363.021,Z 788.346,A -85,B 0,C 180,E1 15638.258,E2 15638.258} C_VEL
LIN {X 0,Y 358.79,Z 807.896,A -85,B 0,C 180,E1 15636.738,E2 15636.738} C_VEL
LIN {X 0,Y 354.487,Z 825.266,A -85,B 0,C 180,E1 15635.076,E2 15635.076} C_VEL
LIN {X 0,Y 349.777,Z 842.176,A -85,B 0,C 180,E1 15633.098,E2 15633.098} C_VEL
LIN {X 0,Y 345.002,Z 857.961,A -85,B 0,C 180,E1 15630.863,E2 15630.863} C_VEL
LIN {X 0,Y 340.368,Z 872.41,A -85,B 0,C 180,E1 15628.409,E2 15628.409} C_VEL
LIN {X 0,Y 335.877,Z 885.994,A -85,B 0,C 180,E1 15625.626,E2 15625.626} C_VEL
LIN {X 0,Y 331.887,Z 897.92,A -85,B 0,C 180,E1 15622.679,E2 15622.679} C_VEL
LIN {X 0,Y 328.167,Z 909.195,A -85,B 0,C 180,E1 15619.245,E2 15619.245} C_VEL
LIN {X 0,Y 325.277,Z 918.385,A -85,B 0,C 180,E1 15615.735,E2 15615.735} C_VEL
LIN {X 0,Y 323.191,Z 925.735,A -85,B 0,C 180,E1 15612.163,E2 15612.163} C_VEL
LIN {X 0,Y 321.768,Z 931.546,A -85,B 0,C 180,E1 15608.418,E2 15608.418} C_VEL
LIN {X 0,Y 320.976,Z 935.58,A -85,B 0,C 180,E1 15604.676,E2 15604.676} C_VEL
LIN {X 0,Y 320.635,Z 937.886,A -85,B 0,C 180,E1 15601.169,E2 15601.169} C_VEL
LIN {X 0,Y 320.497,Z 938.668,A -85,B 0,C 180,E1 15597.624,E2 15597.624} C_VEL
LIN {X 0,Y 320.526,Z 938.043,A -85,B 0,C 180,E1 15594.115,E2 15594.115} C_VEL
LIN {X 0,Y 320.741,Z 936.048,A -85,B 0,C 180,E1 15590.621,E2 15590.621} C_VEL
LIN {X 0,Y 321.277,Z 932.395,A -85,B 0,C 180,E1 15587.006,E2 15587.006} C_VEL
LIN {X 0,Y 322.259,Z 927.18,A -85,B 0,C 180,E1 15583.452,E2 15583.452} C_VEL
LIN {X 0,Y 323.948,Z 919.978,A -85,B 0,C 180,E1 15579.77,E2 15579.77} C_VEL
LIN {X 0,Y 326.263,Z 911.373,A -85,B 0,C 180,E1 15576.33,E2 15576.33} C_VEL
LIN {X 0,Y 329.154,Z 901.492,A -85,B 0,C 180,E1 15573.131,E2 15573.131} C_VEL
LIN {X 0,Y 332.746,Z 889.63,A -85,B 0,C 180,E1 15569.996,E2 15569.996} C_VEL
LIN {X 0,Y 336.792,Z 876.288,A -85,B 0,C 180,E1 15567.104,E2 15567.104} C_VEL
LIN {X 0,Y 340.987,Z 862.146,A -85,B 0,C 180,E1 15564.555,E2 15564.555} C_VEL
LIN {X 0,Y 345.662,Z 845.689,A -85,B 0,C 180,E1 15562.099,E2 15562.099} C_VEL
LIN {X 0,Y 350.03,Z 829.048,A -85,B 0,C 180,E1 15560.045,E2 15560.045} C_VEL
LIN {X 0,Y 354.224,Z 811.651,A -85,B 0,C 180,E1 15558.271,E2 15558.271} C_VEL
LIN {X 0,Y 358.307,Z 792.187,A -85,B 0,C 180,E1 15556.664,E2 15556.664} C_VEL
LIN {X 0,Y 359.844,Z 783.79,A -85,B 0,C 180,E1 15556.078,E2 15556.078} C_VEL
LIN {X 0,Y 360.353,Z 776.867,A -85,B 0,C 180,E1 15555.523,E2 15555.523} C_VEL
LIN {X 0,Y 358.661,Z 759.553,A -85,B 0,C 180,E1 15553.911,E2 15553.911} C_VEL
LIN {X 0,Y 358.871,Z 752.334,A -85,B 0,C 180,E1 15553.468,E2 15553.468} C_VEL
LIN {X 0,Y 361.277,Z 730.687,A -85,B 0,C 180,E1 15552.668,E2 15552.668} C_VEL
LIN {X 0,Y 362.983,Z 705.788,A -85,B 0,C 180,E1 15552.059,E2 15552.059} C_VEL
LIN {X 0,Y 373.092,Z 519.343,A -85,B 0,C 180,E1 15548.188,E2 15548.188} C_VEL
LIN {X 0,Y 362.521,Z 501.356,A -85,B 0,C 180,E1 15545.625,E2 15545.625} C_VEL
LIN {X 0,Y 351.429,Z 484.156,A -85,B 0,C 180,E1 15542.681,E2 15542.681} C_VEL
LIN {X 0,Y 341.435,Z 470.072,A -85,B 0,C 180,E1 15539.753,E2 15539.753} C_VEL
LIN {X 0,Y 334.634,Z 460.894,A -85,B 0,C 180,E1 15537.575,E2 15537.575} C_VEL
LIN {X 0,Y 328.423,Z 452.521,A -85,B 0,C 180,E1 15535.286,E2 15535.286} C_VEL
LIN {X 0,Y 325.183,Z 446.565,A -85,B 0,C 180,E1 15532.937,E2 15532.937} C_VEL
LIN {X 0,Y 322.813,Z 442.025,A -85,B 0,C 180,E1 15531.027,E2 15531.027} C_VEL
LIN {X 0,Y 320.628,Z 438.283,A -85,B 0,C 180,E1 15529.27,E2 15529.27} C_VEL
LIN {X 0,Y 319.563,Z 436.547,A -85,B 0,C 180,E1 15528.4,E2 15528.4} C_VEL
LIN {X 0,Y 317.62,Z 433.116,A -85,B 0,C 180,E1 15526.651,E2 15526.651} C_VEL
LIN {X 0,Y 316.694,Z 431.507,A -85,B 0,C 180,E1 15525.782,E2 15525.782} C_VEL
LIN {X 0,Y 314.578,Z 428.299,A -85,B 0,C 180,E1 15523.818,E2 15523.818} C_VEL
LIN {X 0,Y 314.193,Z 426.777,A -85,B 0,C 180,E1 15522.924,E2 15522.924} C_VEL
LIN {X 0,Y 314.168,Z 426.588,A -85,B 0,C 180,E1 15518.593,E2 15518.593} C_VEL
LIN {X 0,Y 314.174,Z 426.602,A -85,B 0,C 180,E1 15514.065,E2 15514.065} C_VEL
LIN {X 0,Y 314.173,Z 426.581,A -85,B 0,C 180,E1 15509.558,E2 15509.558} C_VEL
LIN {X 0,Y 314.166,Z 426.564,A -85,B 0,C 180,E1 15505.043,E2 15505.043} C_VEL
LIN {X 0,Y 314.167,Z 426.563,A -85,B 0,C 180,E1 15500.656,E2 15500.656} C_VEL
LIN {X 0,Y 314.168,Z 426.582,A -85,B 0,C 180,E1 15496.265,E2 15496.265} C_VEL
LIN {X 0,Y 314.17,Z 426.602,A -85,B 0,C 180,E1 15491.753,E2 15491.753} C_VEL
LIN {X 0,Y 314.178,Z 426.573,A -85,B 0,C 180,E1 15487.314,E2 15487.314} C_VEL
LIN {X 0,Y 314.163,Z 426.563,A -85,B 0,C 180,E1 15482.737,E2 15482.737} C_VEL
LIN {X 0,Y 314.163,Z 426.566,A -85,B 0,C 180,E1 15478.359,E2 15478.359} C_VEL
LIN {X 0,Y 314.169,Z 426.573,A -85,B 0,C 180,E1 15473.789,E2 15473.789} C_VEL
LIN {X 0,Y 314.198,Z 426.83,A -85,B 0,C 180,E1 15470.291,E2 15470.291} C_VEL
LIN {X 0,Y 315.932,Z 430.677,A -85,B 0,C 180,E1 15468.129,E2 15468.129} C_VEL
LIN {X 0,Y 317.544,Z 432.501,A -85,B 0,C 180,E1 15466.897,E2 15466.897} C_VEL
LIN {X 0,Y 319.41,Z 436.268,A -85,B 0,C 180,E1 15465.127,E2 15465.127} C_VEL
LIN {X 0,Y 320.863,Z 438.105,A -85,B 0,C 180,E1 15464.085,E2 15464.085} C_VEL
LIN {X 0,Y 323.01,Z 442.056,A -85,B 0,C 180,E1 15462.341,E2 15462.341} C_VEL
LIN {X 0,Y 323.974,Z 443.583,A -85,B 0,C 180,E1 15461.652,E2 15461.652} C_VEL
LIN {X 0,Y 326.556,Z 447.815,A -85,B 0,C 180,E1 15459.852,E2 15459.852} C_VEL
LIN {X 0,Y 330.095,Z 454.499,A -85,B 0,C 180,E1 15457.423,E2 15457.423} C_VEL
LIN {X 0,Y 338.408,Z 465.21,A -85,B 0,C 180,E1 15454.587,E2 15454.587} C_VEL
LIN {X 0,Y 342.498,Z 470.679,A -85,B 0,C 180,E1 15453.284,E2 15453.284} C_VEL
LIN {X 0,Y 351.2,Z 482.535,A -85,B 0,C 180,E1 15450.728,E2 15450.728} C_VEL
LIN {X 0,Y 362.227,Z 498.801,A -85,B 0,C 180,E1 15447.763,E2 15447.763} C_VEL
LIN {X 0,Y 373.363,Z 516.684,A -85,B 0,C 180,E1 15445.035,E2 15445.035} C_VEL
LIN {X 0,Y 377.972,Z 524.831,A -85,B 0,C 180,E1 15443.96,E2 15443.96} C_VEL
LIN {X 0,Y 366.444,Z 753.132,A -85,B 0,C 180,E1 15439.361,E2 15439.361} C_VEL
LIN {X 0,Y 364.093,Z 775.119,A -85,B 0,C 180,E1 15438.702,E2 15438.702} C_VEL
LIN {X 0,Y 361.014,Z 795.984,A -85,B 0,C 180,E1 15437.838,E2 15437.838} C_VEL
LIN {X 0,Y 357.465,Z 815.849,A -85,B 0,C 180,E1 15436.764,E2 15436.764} C_VEL
LIN {X 0,Y 353.122,Z 835.979,A -85,B 0,C 180,E1 15435.37,E2 15435.37} C_VEL
LIN {X 0,Y 348.264,Z 855.882,A -85,B 0,C 180,E1 15433.658,E2 15433.658} C_VEL
LIN {X 0,Y 343.1,Z 875.031,A -85,B 0,C 180,E1 15431.642,E2 15431.642} C_VEL
LIN {X 0,Y 337.997,Z 892.734,A -85,B 0,C 180,E1 15429.388,E2 15429.388} C_VEL
LIN {X 0,Y 332.87,Z 909.375,A -85,B 0,C 180,E1 15426.819,E2 15426.819} C_VEL
LIN {X 0,Y 327.966,Z 925.1,A -85,B 0,C 180,E1 15423.914,E2 15423.914} C_VEL
LIN {X 0,Y 323.637,Z 939.179,A -85,B 0,C 180,E1 15420.812,E2 15420.812} C_VEL
LIN {X 0,Y 319.803,Z 952.224,A -85,B 0,C 180,E1 15417.364,E2 15417.364} C_VEL
LIN {X 0,Y 316.774,Z 963.453,A -85,B 0,C 180,E1 15413.746,E2 15413.746} C_VEL
LIN {X 0,Y 314.534,Z 973.276,A -85,B 0,C 180,E1 15409.889,E2 15409.889} C_VEL
LIN {X 0,Y 313.149,Z 981.162,A -85,B 0,C 180,E1 15406.042,E2 15406.042} C_VEL
LIN {X 0,Y 312.466,Z 986.961,A -85,B 0,C 180,E1 15402.384,E2 15402.384} C_VEL
LIN {X 0,Y 312.248,Z 991.488,A -85,B 0,C 180,E1 15398.474,E2 15398.474} C_VEL
LIN {X 0,Y 312.258,Z 994.14,A -85,B 0,C 180,E1 15394.963,E2 15394.963} C_VEL
LIN {X 0,Y 312.342,Z 995.361,A -85,B 0,C 180,E1 15391.288,E2 15391.288} C_VEL
LIN {X 0,Y 312.332,Z 995.211,A -85,B 0,C 180,E1 15387.986,E2 15387.986} C_VEL
LIN {X 0,Y 312.265,Z 993.545,A -85,B 0,C 180,E1 15384.308,E2 15384.308} C_VEL
LIN {X 0,Y 312.261,Z 990.591,A -85,B 0,C 180,E1 15380.792,E2 15380.792} C_VEL
LIN {X 0,Y 312.54,Z 985.907,A -85,B 0,C 180,E1 15377.064,E2 15377.064} C_VEL
LIN {X 0,Y 313.326,Z 979.702,A -85,B 0,C 180,E1 15373.314,E2 15373.314} C_VEL
LIN {X 0,Y 314.782,Z 971.668,A -85,B 0,C 180,E1 15369.554,E2 15369.554} C_VEL
LIN {X 0,Y 317.208,Z 961.315,A -85,B 0,C 180,E1 15365.617,E2 15365.617} C_VEL
LIN {X 0,Y 320.366,Z 949.878,A -85,B 0,C 180,E1 15362.035,E2 15362.035} C_VEL
LIN {X 0,Y 324.354,Z 936.723,A -85,B 0,C 180,E1 15358.609,E2 15358.609} C_VEL
LIN {X 0,Y 328.795,Z 922.639,A -85,B 0,C 180,E1 15355.56,E2 15355.56} C_VEL
LIN {X 0,Y 334.03,Z 906.282,A -85,B 0,C 180,E1 15352.587,E2 15352.587} C_VEL
LIN {X 0,Y 339.35,Z 889.495,A -85,B 0,C 180,E1 15350.042,E2 15350.042} C_VEL
LIN {X 0,Y 344.548,Z 872.094,A -85,B 0,C 180,E1 15347.849,E2 15347.849} C_VEL
LIN {X 0,Y 349.799,Z 853.392,A -85,B 0,C 180,E1 15345.898,E2 15345.898} C_VEL
LIN {X 0,Y 354.888,Z 833.455,A -85,B 0,C 180,E1 15344.197,E2 15344.197} C_VEL
LIN {X 0,Y 359.306,Z 813.822,A -85,B 0,C 180,E1 15342.847,E2 15342.847} C_VEL
LIN {X 0,Y 363.156,Z 793.442,A -85,B 0,C 180,E1 15341.751,E2 15341.751} C_VEL
LIN {X 0,Y 366.583,Z 771.087,A -85,B 0,C 180,E1 15340.847,E2 15340.847} C_VEL
LIN {X 0,Y 368.953,Z 749.25,A -85,B 0,C 180,E1 15340.215,E2 15340.215} C_VEL
LIN {X 0,Y 381.586,Z 524.919,A -85,B 0,C 180,E1 15335.606,E2 15335.606} C_VEL
LIN {X 0,Y 373.689,Z 510.691,A -85,B 0,C 180,E1 15333.264,E2 15333.264} C_VEL
LIN {X 0,Y 366.977,Z 499.704,A -85,B 0,C 180,E1 15331.039,E2 15331.039} C_VEL
LIN {X 0,Y 360.676,Z 490.244,A -85,B 0,C 180,E1 15328.658,E2 15328.658} C_VEL
LIN {X 0,Y 355.478,Z 482.859,A -85,B 0,C 180,E1 15326.385,E2 15326.385} C_VEL
LIN {X 0,Y 351.821,Z 477.928,A -85,B 0,C 180,E1 15324.514,E2 15324.514} C_VEL
LIN {X 0,Y 348.694,Z 473.742,A -85,B 0,C 180,E1 15322.685,E2 15322.685} C_VEL
LIN {X 0,Y 344.807,Z 468.647,A -85,B 0,C 180,E1 15319.832,E2 15319.832} C_VEL
LIN {X 0,Y 340.519,Z 463.267,A -85,B 0,C 180,E1 15314.452,E2 15314.452} C_VEL
LIN {X 0,Y 339.689,Z 462.591,A -85,B 0,C 180,E1 15310.686,E2 15310.686} C_VEL
LIN {X 0,Y 340.519,Z 463.336,A -85,B 0,C 180,E1 15307.423,E2 15307.423} C_VEL
LIN {X 0,Y 344.963,Z 469.122,A -85,B 0,C 180,E1 15301.91,E2 15301.91} C_VEL
LIN {X 0,Y 349.288,Z 474.986,A -85,B 0,C 180,E1 15298.769,E2 15298.769} C_VEL
LIN {X 0,Y 353.021,Z 480.149,A -85,B 0,C 180,E1 15296.63,E2 15296.63} C_VEL
LIN {X 0,Y 356.087,Z 484.326,A -85,B 0,C 180,E1 15295.123,E2 15295.123} C_VEL
LIN {X 0,Y 360.637,Z 490.974,A -85,B 0,C 180,E1 15293.113,E2 15293.113} C_VEL
LIN {X 0,Y 366.804,Z 500.382,A -85,B 0,C 180,E1 15290.745,E2 15290.745} C_VEL
LIN {X 0,Y 373.785,Z 512.063,A -85,B 0,C 180,E1 15288.387,E2 15288.387} C_VEL
LIN {X 0,Y 380.065,Z 523.437,A -85,B 0,C 180,E1 15286.476,E2 15286.476} C_VEL
LIN {X 0,Y 366.621,Z 727.583,A -85,B 0,C 180,E1 15282.087,E2 15282.087} C_VEL
LIN {X 0,Y 364.328,Z 748.344,A -85,B 0,C 180,E1 15281.379,E2 15281.379} C_VEL
LIN {X 0,Y 361.31,Z 768.443,A -85,B 0,C 180,E1 15280.436,E2 15280.436} C_VEL
LIN {X 0,Y 357.522,Z 788.641,A -85,B 0,C 180,E1 15279.195,E2 15279.195} C_VEL
LIN {X 0,Y 353.233,Z 807.734,A -85,B 0,C 180,E1 15277.709,E2 15277.709} C_VEL
LIN {X 0,Y 348.544,Z 825.869,A -85,B 0,C 180,E1 15275.961,E2 15275.961} C_VEL
LIN {X 0,Y 343.386,Z 843.607,A -85,B 0,C 180,E1 15273.858,E2 15273.858} C_VEL
LIN {X 0,Y 338.3,Z 859.58,A -85,B 0,C 180,E1 15271.544,E2 15271.544} C_VEL
LIN {X 0,Y 333.437,Z 873.911,A -85,B 0,C 180,E1 15269.039,E2 15269.039} C_VEL
LIN {X 0,Y 328.65,Z 887.622,A -85,B 0,C 180,E1 15266.146,E2 15266.146} C_VEL
LIN {X 0,Y 324.366,Z 899.687,A -85,B 0,C 180,E1 15263.052,E2 15263.052} C_VEL
LIN {X 0,Y 320.619,Z 910.439,A -85,B 0,C 180,E1 15259.665,E2 15259.665} C_VEL
LIN {X 0,Y 317.615,Z 919.44,A -85,B 0,C 180,E1 15256.121,E2 15256.121} C_VEL
LIN {X 0,Y 315.403,Z 926.704,A -85,B 0,C 180,E1 15252.465,E2 15252.465} C_VEL
LIN {X 0,Y 313.909,Z 932.337,A -85,B 0,C 180,E1 15248.705,E2 15248.705} C_VEL
LIN {X 0,Y 313.043,Z 936.377,A -85,B 0,C 180,E1 15244.828,E2 15244.828} C_VEL
LIN {X 0,Y 312.673,Z 938.652,A -85,B 0,C 180,E1 15241.195,E2 15241.195} C_VEL
LIN {X 0,Y 312.529,Z 939.396,A -85,B 0,C 180,E1 15237.6,E2 15237.6} C_VEL
LIN {X 0,Y 312.562,Z 938.718,A -85,B 0,C 180,E1 15233.965,E2 15233.965} C_VEL
LIN {X 0,Y 312.807,Z 936.67,A -85,B 0,C 180,E1 15230.385,E2 15230.385} C_VEL
LIN {X 0,Y 313.388,Z 932.993,A -85,B 0,C 180,E1 15226.682,E2 15226.682} C_VEL
LIN {X 0,Y 314.461,Z 927.73,A -85,B 0,C 180,E1 15223.043,E2 15223.043} C_VEL
LIN {X 0,Y 316.206,Z 920.757,A -85,B 0,C 180,E1 15219.401,E2 15219.401} C_VEL
LIN {X 0,Y 318.756,Z 911.824,A -85,B 0,C 180,E1 15215.757,E2 15215.757} C_VEL
LIN {X 0,Y 321.829,Z 901.888,A -85,B 0,C 180,E1 15212.489,E2 15212.489} C_VEL
LIN {X 0,Y 325.637,Z 889.982,A -85,B 0,C 180,E1 15209.293,E2 15209.293} C_VEL
LIN {X 0,Y 329.901,Z 876.563,A -85,B 0,C 180,E1 15206.347,E2 15206.347} C_VEL
LIN {X 0,Y 334.353,Z 862.171,A -85,B 0,C 180,E1 15203.73,E2 15203.73} C_VEL
LIN {X 0,Y 339.195,Z 845.777,A -85,B 0,C 180,E1 15201.265,E2 15201.265} C_VEL
LIN {X 0,Y 343.94,Z 828.311,A -85,B 0,C 180,E1 15199.105,E2 15199.105} C_VEL
LIN {X 0,Y 348.322,Z 810.623,A -85,B 0,C 180,E1 15197.312,E2 15197.312} C_VEL
LIN {X 0,Y 352.326,Z 792.194,A -85,B 0,C 180,E1 15195.787,E2 15195.787} C_VEL
LIN {X 0,Y 355.932,Z 772.309,A -85,B 0,C 180,E1 15194.48,E2 15194.48} C_VEL
LIN {X 0,Y 358.871,Z 752.334,A -85,B 0,C 180,E1 15193.468,E2 15193.468} C_VEL
LIN {X 0,Y 359.16,Z 746.047,A -85,B 0,C 180,E1 15193.117,E2 15193.117} C_VEL
LIN {X 0,Y 356.694,Z 726.757,A -85,B 0,C 180,E1 15191.755,E2 15191.755} C_VEL
LIN {X 0,Y 356.546,Z 719.255,A -85,B 0,C 180,E1 15191.448,E2 15191.448} C_VEL
LIN {X 0,Y 367.716,Z 522.865,A -85,B 0,C 180,E1 15187.317,E2 15187.317} C_VEL
LIN {X 0,Y 358.02,Z 506.293,A -85,B 0,C 180,E1 15184.878,E2 15184.878} C_VEL
LIN {X 0,Y 347.667,Z 490.118,A -85,B 0,C 180,E1 15182.042,E2 15182.042} C_VEL
LIN {X 0,Y 338.01,Z 476.306,A -85,B 0,C 180,E1 15179.121,E2 15179.121} C_VEL
LIN {X 0,Y 329.97,Z 465.374,A -85,B 0,C 180,E1 15176.439,E2 15176.439} C_VEL
LIN {X 0,Y 324.002,Z 457.762,A -85,B 0,C 180,E1 15174.254,E2 15174.254} C_VEL
LIN {X 0,Y 320.349,Z 452.836,A -85,B 0,C 180,E1 15172.732,E2 15172.732} C_VEL
LIN {X 0,Y 317.83,Z 448.121,A -85,B 0,C 180,E1 15170.705,E2 15170.705} C_VEL
LIN {X 0,Y 315.596,Z 443.923,A -85,B 0,C 180,E1 15168.775,E2 15168.775} C_VEL
LIN {X 0,Y 312.973,Z 439.644,A -85,B 0,C 180,E1 15166.486,E2 15166.486} C_VEL
LIN {X 0,Y 312.092,Z 437.988,A -85,B 0,C 180,E1 15165.597,E2 15165.597} C_VEL
LIN {X 0,Y 309.86,Z 434.402,A -85,B 0,C 180,E1 15163.418,E2 15163.418} C_VEL
LIN {X 0,Y 309.04,Z 432.774,A -85,B 0,C 180,E1 15162.463,E2 15162.463} C_VEL
LIN {X 0,Y 306.562,Z 429.045,A -85,B 0,C 180,E1 15159.737,E2 15159.737} C_VEL
LIN {X 0,Y 306.251,Z 427.74,A -85,B 0,C 180,E1 15158.708,E2 15158.708} C_VEL
LIN {X 0,Y 306.236,Z 427.588,A -85,B 0,C 180,E1 15154.166,E2 15154.166} C_VEL
LIN {X 0,Y 306.234,Z 427.568,A -85,B 0,C 180,E1 15149.54,E2 15149.54} C_VEL
LIN {X 0,Y 306.227,Z 427.551,A -85,B 0,C 180,E1 15145.117,E2 15145.117} C_VEL
LIN {X 0,Y 306.229,Z 427.55,A -85,B 0,C 180,E1 15140.649,E2 15140.649} C_VEL
LIN {X 0,Y 306.228,Z 427.566,A -85,B 0,C 180,E1 15136.114,E2 15136.114} C_VEL
LIN {X 0,Y 306.233,Z 427.591,A -85,B 0,C 180,E1 15131.489,E2 15131.489} C_VEL
LIN {X 0,Y 306.231,Z 427.568,A -85,B 0,C 180,E1 15126.939,E2 15126.939} C_VEL
LIN {X 0,Y 306.224,Z 427.554,A -85,B 0,C 180,E1 15122.342,E2 15122.342} C_VEL
LIN {X 0,Y 306.226,Z 427.552,A -85,B 0,C 180,E1 15117.942,E2 15117.942} C_VEL
LIN {X 0,Y 306.272,Z 427.893,A -85,B 0,C 180,E1 15114.38,E2 15114.38} C_VEL
LIN {X 0,Y 308.287,Z 431.995,A -85,B 0,C 180,E1 15111.608,E2 15111.608} C_VEL
LIN {X 0,Y 309.699,Z 433.595,A -85,B 0,C 180,E1 15110.336,E2 15110.336} C_VEL
LIN {X 0,Y 311.744,Z 437.524,A -85,B 0,C 180,E1 15108.155,E2 15108.155} C_VEL
LIN {X 0,Y 313.063,Z 439.169,A -85,B 0,C 180,E1 15107.082,E2 15107.082} C_VEL
LIN {X 0,Y 315.219,Z 443.154,A -85,B 0,C 180,E1 15105.113,E2 15105.113} C_VEL
LIN {X 0,Y 316.346,Z 444.827,A -85,B 0,C 180,E1 15104.228,E2 15104.228} C_VEL
LIN {X 0,Y 318.806,Z 448.961,A -85,B 0,C 180,E1 15102.289,E2 15102.289} C_VEL
LIN {X 0,Y 321.651,Z 453.945,A -85,B 0,C 180,E1 15100.195,E2 15100.195} C_VEL
LIN {X 0,Y 325.998,Z 459.554,A -85,B 0,C 180,E1 15098.453,E2 15098.453} C_VEL
LIN {X 0,Y 337.926,Z 475.076,A -85,B 0,C 180,E1 15094.313,E2 15094.313} C_VEL
LIN {X 0,Y 348.855,Z 490.527,A -85,B 0,C 180,E1 15090.982,E2 15090.982} C_VEL
LIN {X 0,Y 358.631,Z 505.139,A -85,B 0,C 180,E1 15088.296,E2 15088.296} C_VEL
LIN {X 0,Y 369.445,Z 522.71,A -85,B 0,C 180,E1 15085.578,E2 15085.578} C_VEL
LIN {X 0,Y 372.591,Z 528.329,A -85,B 0,C 180,E1 15084.823,E2 15084.823} C_VEL
LIN {X 0,Y 360.769,Z 752.899,A -85,B 0,C 180,E1 15080.255,E2 15080.255} C_VEL
LIN {X 0,Y 358.325,Z 775.058,A -85,B 0,C 180,E1 15079.585,E2 15079.585} C_VEL
LIN {X 0,Y 355.083,Z 796.23,A -85,B 0,C 180,E1 15078.698,E2 15078.698} C_VEL
LIN {X 0,Y 351.308,Z 816.475,A -85,B 0,C 180,E1 15077.583,E2 15077.583} C_VEL
LIN {X 0,Y 346.952,Z 835.999,A -85,B 0,C 180,E1 15076.215,E2 15076.215} C_VEL
LIN {X 0,Y 342.089,Z 855.154,A -85,B 0,C 180,E1 15074.548,E2 15074.548} C_VEL
LIN {X 0,Y 336.901,Z 873.717,A -85,B 0,C 180,E1 15072.586,E2 15072.586} C_VEL
LIN {X 0,Y 331.456,Z 891.865,A -85,B 0,C 180,E1 15070.254,E2 15070.254} C_VEL
LIN {X 0,Y 326.307,Z 907.891,A -85,B 0,C 180,E1 15067.764,E2 15067.764} C_VEL
LIN {X 0,Y 321.043,Z 924.089,A -85,B 0,C 180,E1 15064.749,E2 15064.749} C_VEL
LIN {X 0,Y 316.512,Z 938.069,A -85,B 0,C 180,E1 15061.631,E2 15061.631} C_VEL
LIN {X 0,Y 312.582,Z 950.637,A -85,B 0,C 180,E1 15058.259,E2 15058.259} C_VEL
LIN {X 0,Y 309.365,Z 961.81,A -85,B 0,C 180,E1 15054.644,E2 15054.644} C_VEL
LIN {X 0,Y 306.938,Z 971.636,A -85,B 0,C 180,E1 15050.788,E2 15050.788} C_VEL
LIN {X 0,Y 305.396,Z 979.542,A -85,B 0,C 180,E1 15046.944,E2 15046.944} C_VEL
LIN {X 0,Y 304.561,Z 985.657,A -85,B 0,C 180,E1 15043.096,E2 15043.096} C_VEL
LIN {X 0,Y 304.267,Z 990.236,A -85,B 0,C 180,E1 15039.27,E2 15039.27} C_VEL
LIN {X 0,Y 304.283,Z 993.056,A -85,B 0,C 180,E1 15035.661,E2 15035.661} C_VEL
LIN {X 0,Y 304.36,Z 994.58,A -85,B 0,C 180,E1 15031.887,E2 15031.887} C_VEL
LIN {X 0,Y 304.373,Z 994.587,A -85,B 0,C 180,E1 15028.498,E2 15028.498} C_VEL
LIN {X 0,Y 304.288,Z 993.21,A -85,B 0,C 180,E1 15024.725,E2 15024.725} C_VEL
LIN {X 0,Y 304.274,Z 990.403,A -85,B 0,C 180,E1 15021.12,E2 15021.12} C_VEL
LIN {X 0,Y 304.538,Z 985.729,A -85,B 0,C 180,E1 15017.104,E2 15017.104} C_VEL
LIN {X 0,Y 305.332,Z 979.641,A -85,B 0,C 180,E1 15013.256,E2 15013.256} C_VEL
LIN {X 0,Y 306.827,Z 971.802,A -85,B 0,C 180,E1 15009.399,E2 15009.399} C_VEL
LIN {X 0,Y 309.194,Z 962.207,A -85,B 0,C 180,E1 15005.554,E2 15005.554} C_VEL
LIN {X 0,Y 312.557,Z 950.645,A -85,B 0,C 180,E1 15001.747,E2 15001.747} C_VEL
LIN {X 0,Y 316.493,Z 938.194,A -85,B 0,C 180,E1 14998.376,E2 14998.376} C_VEL
LIN {X 0,Y 321.343,Z 923.683,A -85,B 0,C 180,E1 14995.08,E2 14995.08} C_VEL
LIN {X 0,Y 326.472,Z 908.559,A -85,B 0,C 180,E1 14992.199,E2 14992.199} C_VEL
LIN {X 0,Y 332.253,Z 891.199,A -85,B 0,C 180,E1 14989.464,E2 14989.464} C_VEL
LIN {X 0,Y 337.705,Z 873.892,A -85,B 0,C 180,E1 14987.203,E2 14987.203} C_VEL
LIN {X 0,Y 343.482,Z 854.395,A -85,B 0,C 180,E1 14985.104,E2 14985.104} C_VEL
LIN {X 0,Y 348.831,Z 834.538,A -85,B 0,C 180,E1 14983.364,E2 14983.364} C_VEL
LIN {X 0,Y 353.564,Z 814.418,A -85,B 0,C 180,E1 14981.956,E2 14981.956} C_VEL
LIN {X 0,Y 357.682,Z 793.673,A -85,B 0,C 180,E1 14980.82,E2 14980.82} C_VEL
LIN {X 0,Y 361.156,Z 772.165,A -85,B 0,C 180,E1 14979.934,E2 14979.934} C_VEL
LIN {X 0,Y 363.736,Z 749.934,A -85,B 0,C 180,E1 14979.272,E2 14979.272} C_VEL
LIN {X 0,Y 376.845,Z 528.798,A -85,B 0,C 180,E1 14974.681,E2 14974.681} C_VEL
LIN {X 0,Y 370.198,Z 516.549,A -85,B 0,C 180,E1 14972.603,E2 14972.603} C_VEL
LIN {X 0,Y 363.914,Z 505.993,A -85,B 0,C 180,E1 14970.412,E2 14970.412} C_VEL
LIN {X 0,Y 357.348,Z 495.697,A -85,B 0,C 180,E1 14967.766,E2 14967.766} C_VEL
LIN {X 0,Y 352.853,Z 489.43,A -85,B 0,C 180,E1 14965.692,E2 14965.692} C_VEL
LIN {X 0,Y 349.786,Z 485.131,A -85,B 0,C 180,E1 14964.037,E2 14964.037} C_VEL
LIN {X 0,Y 346.922,Z 481.187,A -85,B 0,C 180,E1 14962.271,E2 14962.271} C_VEL
LIN {X 0,Y 343.384,Z 476.373,A -85,B 0,C 180,E1 14959.563,E2 14959.563} C_VEL
LIN {X 0,Y 339.38,Z 471.156,A -85,B 0,C 180,E1 14954.328,E2 14954.328} C_VEL
LIN {X 0,Y 338.611,Z 470.525,A -85,B 0,C 180,E1 14950.518,E2 14950.518} C_VEL
LIN {X 0,Y 339.409,Z 471.326,A -85,B 0,C 180,E1 14947.447,E2 14947.447} C_VEL
LIN {X 0,Y 343.418,Z 476.704,A -85,B 0,C 180,E1 14942.252,E2 14942.252} C_VEL
LIN {X 0,Y 347.714,Z 482.752,A -85,B 0,C 180,E1 14939.011,E2 14939.011} C_VEL
LIN {X 0,Y 351.156,Z 487.652,A -85,B 0,C 180,E1 14936.98,E2 14936.98} C_VEL
LIN {X 0,Y 354.11,Z 491.861,A -85,B 0,C 180,E1 14935.465,E2 14935.465} C_VEL
LIN {X 0,Y 359.127,Z 499.311,A -85,B 0,C 180,E1 14933.204,E2 14933.204} C_VEL
LIN {X 0,Y 366.233,Z 510.767,A -85,B 0,C 180,E1 14930.453,E2 14930.453} C_VEL
LIN {X 0,Y 373.377,Z 523.478,A -85,B 0,C 180,E1 14928.041,E2 14928.041} C_VEL
LIN {X 0,Y 375.356,Z 527.523,A -85,B 0,C 180,E1 14927.405,E2 14927.405} C_VEL
LIN {X 0,Y 361.549,Z 728.19,A -85,B 0,C 180,E1 14923.056,E2 14923.056} C_VEL
LIN {X 0,Y 359.157,Z 749.047,A -85,B 0,C 180,E1 14922.34,E2 14922.34} C_VEL
LIN {X 0,Y 355.996,Z 769.239,A -85,B 0,C 180,E1 14921.384,E2 14921.384} C_VEL
LIN {X 0,Y 351.937,Z 789.865,A -85,B 0,C 180,E1 14920.099,E2 14920.099} C_VEL
LIN {X 0,Y 347.341,Z 809.325,A -85,B 0,C 180,E1 14918.556,E2 14918.556} C_VEL
LIN {X 0,Y 342.456,Z 827.344,A -85,B 0,C 180,E1 14916.786,E2 14916.786} C_VEL
LIN {X 0,Y 337.229,Z 844.524,A -85,B 0,C 180,E1 14914.717,E2 14914.717} C_VEL
LIN {X 0,Y 331.841,Z 860.632,A -85,B 0,C 180,E1 14912.344,E2 14912.344} C_VEL
LIN {X 0,Y 326.801,Z 874.79,A -85,B 0,C 180,E1 14909.826,E2 14909.826} C_VEL
LIN {X 0,Y 321.556,Z 888.987,A -85,B 0,C 180,E1 14906.756,E2 14906.756} C_VEL
LIN {X 0,Y 316.984,Z 901.143,A -85,B 0,C 180,E1 14903.538,E2 14903.538} C_VEL
LIN {X 0,Y 313.262,Z 911.23,A -85,B 0,C 180,E1 14900.275,E2 14900.275} C_VEL
LIN {X 0,Y 309.969,Z 920.496,A -85,B 0,C 180,E1 14896.526,E2 14896.526} C_VEL
LIN {X 0,Y 307.595,Z 927.781,A -85,B 0,C 180,E1 14892.723,E2 14892.723} C_VEL
LIN {X 0,Y 306.045,Z 933.196,A -85,B 0,C 180,E1 14888.962,E2 14888.962} C_VEL
LIN {X 0,Y 305.113,Z 937.177,A -85,B 0,C 180,E1 14884.987,E2 14884.987} C_VEL
LIN {X 0,Y 304.711,Z 939.415,A -85,B 0,C 180,E1 14881.223,E2 14881.223} C_VEL
LIN {X 0,Y 304.562,Z 940.122,A -85,B 0,C 180,E1 14877.569,E2 14877.569} C_VEL
LIN {X 0,Y 304.599,Z 939.391,A -85,B 0,C 180,E1 14873.808,E2 14873.808} C_VEL
LIN {X 0,Y 304.896,Z 937.121,A -85,B 0,C 180,E1 14869.936,E2 14869.936} C_VEL
LIN {X 0,Y 305.553,Z 933.357,A -85,B 0,C 180,E1 14866.145,E2 14866.145} C_VEL
LIN {X 0,Y 306.837,Z 927.66,A -85,B 0,C 180,E1 14862.224,E2 14862.224} C_VEL
LIN {X 0,Y 308.755,Z 920.568,A -85,B 0,C 180,E1 14858.563,E2 14858.563} C_VEL
LIN {X 0,Y 311.442,Z 911.75,A -85,B 0,C 180,E1 14854.969,E2 14854.969} C_VEL
LIN {X 0,Y 314.948,Z 901.006,A -85,B 0,C 180,E1 14851.451,E2 14851.451} C_VEL
LIN {X 0,Y 318.814,Z 889.547,A -85,B 0,C 180,E1 14848.379,E2 14848.379} C_VEL
LIN {X 0,Y 323.354,Z 875.985,A -85,B 0,C 180,E1 14845.385,E2 14845.385} C_VEL
LIN {X 0,Y 328.236,Z 860.848,A -85,B 0,C 180,E1 14842.646,E2 14842.646} C_VEL
LIN {X 0,Y 332.979,Z 845.265,A -85,B 0,C 180,E1 14840.316,E2 14840.316} C_VEL
LIN {X 0,Y 337.76,Z 828.269,A -85,B 0,C 180,E1 14838.211,E2 14838.211} C_VEL
LIN {X 0,Y 342.319,Z 810.426,A -85,B 0,C 180,E1 14836.398,E2 14836.398} C_VEL
LIN {X 0,Y 346.481,Z 791.849,A -85,B 0,C 180,E1 14834.858,E2 14834.858} C_VEL
LIN {X 0,Y 350.28,Z 771.455,A -85,B 0,C 180,E1 14833.522,E2 14833.522} C_VEL
LIN {X 0,Y 353.387,Z 750.667,A -85,B 0,C 180,E1 14832.487,E2 14832.487} C_VEL
LIN {X 0,Y 355.693,Z 729.909,A -85,B 0,C 180,E1 14831.736,E2 14831.736} C_VEL
LIN {X 0,Y 356.546,Z 719.255,A -85,B 0,C 180,E1 14831.448,E2 14831.448} C_VEL
LIN {X 0,Y 356.362,Z 711.703,A -85,B 0,C 180,E1 14831.159,E2 14831.159} C_VEL
LIN {X 0,Y 353.185,Z 691.945,A -85,B 0,C 180,E1 14830.005,E2 14830.005} C_VEL
LIN {X 0,Y 353.035,Z 685.437,A -85,B 0,C 180,E1 14829.776,E2 14829.776} C_VEL
LIN {X 0,Y 362.359,Z 526.322,A -85,B 0,C 180,E1 14826.413,E2 14826.413} C_VEL
LIN {X 0,Y 353.407,Z 511.022,A -85,B 0,C 180,E1 14824.072,E2 14824.072} C_VEL
LIN {X 0,Y 344.025,Z 496.183,A -85,B 0,C 180,E1 14821.413,E2 14821.413} C_VEL
LIN {X 0,Y 334.455,Z 482.321,A -85,B 0,C 180,E1 14818.432,E2 14818.432} C_VEL
LIN {X 0,Y 325.923,Z 470.585,A -85,B 0,C 180,E1 14815.457,E2 14815.457} C_VEL
LIN {X 0,Y 321.037,Z 464.385,A -85,B 0,C 180,E1 14813.62,E2 14813.62} C_VEL
LIN {X 0,Y 317.34,Z 459.579,A -85,B 0,C 180,E1 14812.117,E2 14812.117} C_VEL
LIN {X 0,Y 312.346,Z 453.4,A -85,B 0,C 180,E1 14809.914,E2 14809.914} C_VEL
LIN {X 0,Y 310.272,Z 449.474,A -85,B 0,C 180,E1 14808.109,E2 14808.109} C_VEL
LIN {X 0,Y 308.11,Z 445.502,A -85,B 0,C 180,E1 14806.012,E2 14806.012} C_VEL
LIN {X 0,Y 305.126,Z 440.425,A -85,B 0,C 180,E1 14802.969,E2 14802.969} C_VEL
LIN {X 0,Y 304.083,Z 438.854,A -85,B 0,C 180,E1 14801.874,E2 14801.874} C_VEL
LIN {X 0,Y 301.906,Z 435.05,A -85,B 0,C 180,E1 14799.194,E2 14799.194} C_VEL
LIN {X 0,Y 300.661,Z 433.302,A -85,B 0,C 180,E1 14797.672,E2 14797.672} C_VEL
LIN {X 0,Y 298.365,Z 429.038,A -85,B 0,C 180,E1 14793.858,E2 14793.858} C_VEL
LIN {X 0,Y 298.292,Z 428.54,A -85,B 0,C 180,E1 14790.891,E2 14790.891} C_VEL
LIN {X 0,Y 298.29,Z 428.54,A -85,B 0,C 180,E1 14786.476,E2 14786.476} C_VEL
LIN {X 0,Y 298.297,Z 428.551,A -85,B 0,C 180,E1 14781.795,E2 14781.795} C_VEL
LIN {X 0,Y 298.293,Z 428.578,A -85,B 0,C 180,E1 14777.156,E2 14777.156} C_VEL
LIN {X 0,Y 298.291,Z 428.557,A -85,B 0,C 180,E1 14772.585,E2 14772.585} C_VEL
LIN {X 0,Y 298.291,Z 428.542,A -85,B 0,C 180,E1 14767.9,E2 14767.9} C_VEL
LIN {X 0,Y 298.285,Z 428.538,A -85,B 0,C 180,E1 14763.267,E2 14763.267} C_VEL
LIN {X 0,Y 298.358,Z 428.984,A -85,B 0,C 180,E1 14759.617,E2 14759.617} C_VEL
LIN {X 0,Y 300.647,Z 433.309,A -85,B 0,C 180,E1 14755.805,E2 14755.805} C_VEL
LIN {X 0,Y 301.969,Z 434.927,A -85,B 0,C 180,E1 14754.3,E2 14754.3} C_VEL
LIN {X 0,Y 304.283,Z 439.007,A -85,B 0,C 180,E1 14751.497,E2 14751.497} C_VEL
LIN {X 0,Y 305.4,Z 440.561,A -85,B 0,C 180,E1 14750.389,E2 14750.389} C_VEL
LIN {X 0,Y 307.749,Z 444.592,A -85,B 0,C 180,E1 14747.999,E2 14747.999} C_VEL
LIN {X 0,Y 308.616,Z 445.92,A -85,B 0,C 180,E1 14747.219,E2 14747.219} C_VEL
LIN {X 0,Y 311.012,Z 450.014,A -85,B 0,C 180,E1 14745.097,E2 14745.097} C_VEL
LIN {X 0,Y 313.939,Z 454.941,A -85,B 0,C 180,E1 14742.867,E2 14742.867} C_VEL
LIN {X 0,Y 320.031,Z 462.446,A -85,B 0,C 180,E1 14740.281,E2 14740.281} C_VEL
LIN {X 0,Y 327.796,Z 472.367,A -85,B 0,C 180,E1 14737.304,E2 14737.304} C_VEL
LIN {X 0,Y 336.241,Z 483.807,A -85,B 0,C 180,E1 14734.411,E2 14734.411} C_VEL
LIN {X 0,Y 345.157,Z 496.457,A -85,B 0,C 180,E1 14731.636,E2 14731.636} C_VEL
LIN {X 0,Y 354.932,Z 511.256,A -85,B 0,C 180,E1 14728.874,E2 14728.874} C_VEL
LIN {X 0,Y 365.544,Z 528.733,A -85,B 0,C 180,E1 14726.131,E2 14726.131} C_VEL
LIN {X 0,Y 367.247,Z 532.098,A -85,B 0,C 180,E1 14725.7,E2 14725.7} C_VEL
LIN {X 0,Y 355.191,Z 752.491,A -85,B 0,C 180,E1 14721.181,E2 14721.181} C_VEL
LIN {X 0,Y 352.676,Z 774.632,A -85,B 0,C 180,E1 14720.507,E2 14720.507} C_VEL
LIN {X 0,Y 349.404,Z 795.405,A -85,B 0,C 180,E1 14719.636,E2 14719.636} C_VEL
LIN {X 0,Y 345.579,Z 815.379,A -85,B 0,C 180,E1 14718.538,E2 14718.538} C_VEL
LIN {X 0,Y 340.994,Z 835.3,A -85,B 0,C 180,E1 14717.136,E2 14717.136} C_VEL
LIN {X 0,Y 335.973,Z 854.457,A -85,B 0,C 180,E1 14715.463,E2 14715.463} C_VEL
LIN {X 0,Y 330.8,Z 872.386,A -85,B 0,C 180,E1 14713.565,E2 14713.565} C_VEL
LIN {X 0,Y 325.227,Z 890.229,A -85,B 0,C 180,E1 14711.261,E2 14711.261} C_VEL
LIN {X 0,Y 319.781,Z 906.581,A -85,B 0,C 180,E1 14708.711,E2 14708.711} C_VEL
LIN {X 0,Y 314.48,Z 922.145,A -85,B 0,C 180,E1 14705.807,E2 14705.807} C_VEL
LIN {X 0,Y 309.66,Z 936.355,A -85,B 0,C 180,E1 14702.634,E2 14702.634} C_VEL
LIN {X 0,Y 305.442,Z 949.05,A -85,B 0,C 180,E1 14699.196,E2 14699.196} C_VEL
LIN {X 0,Y 301.959,Z 960.394,A -85,B 0,C 180,E1 14695.5,E2 14695.5} C_VEL
LIN {X 0,Y 299.418,Z 969.917,A -85,B 0,C 180,E1 14691.76,E2 14691.76} C_VEL
LIN {X 0,Y 297.657,Z 977.991,A -85,B 0,C 180,E1 14687.803,E2 14687.803} C_VEL
LIN {X 0,Y 296.649,Z 984.619,A -85,B 0,C 180,E1 14683.651,E2 14683.651} C_VEL
LIN {X 0,Y 296.289,Z 989.322,A -85,B 0,C 180,E1 14679.718,E2 14679.718} C_VEL
LIN {X 0,Y 296.303,Z 992.205,A -85,B 0,C 180,E1 14676.009,E2 14676.009} C_VEL
LIN {X 0,Y 296.376,Z 993.814,A -85,B 0,C 180,E1 14672.324,E2 14672.324} C_VEL
LIN {X 0,Y 296.406,Z 993.93,A -85,B 0,C 180,E1 14668.844,E2 14668.844} C_VEL
LIN {X 0,Y 296.327,Z 992.881,A -85,B 0,C 180,E1 14665.359,E2 14665.359} C_VEL
LIN {X 0,Y 296.288,Z 990.157,A -85,B 0,C 180,E1 14661.399,E2 14661.399} C_VEL
LIN {X 0,Y 296.488,Z 986.069,A -85,B 0,C 180,E1 14657.54,E2 14657.54} C_VEL
LIN {X 0,Y 297.266,Z 980.005,A -85,B 0,C 180,E1 14653.454,E2 14653.454} C_VEL
LIN {X 0,Y 298.875,Z 971.937,A -85,B 0,C 180,E1 14649.235,E2 14649.235} C_VEL
LIN {X 0,Y 301.326,Z 962.577,A -85,B 0,C 180,E1 14645.291,E2 14645.291} C_VEL
LIN {X 0,Y 304.806,Z 951.13,A -85,B 0,C 180,E1 14641.39,E2 14641.39} C_VEL
LIN {X 0,Y 309.143,Z 938.221,A -85,B 0,C 180,E1 14637.753,E2 14637.753} C_VEL
LIN {X 0,Y 314.219,Z 923.865,A -85,B 0,C 180,E1 14634.393,E2 14634.393} C_VEL
LIN {X 0,Y 319.594,Z 908.86,A -85,B 0,C 180,E1 14631.455,E2 14631.455} C_VEL
LIN {X 0,Y 325.386,Z 892.268,A -85,B 0,C 180,E1 14628.773,E2 14628.773} C_VEL
LIN {X 0,Y 331.144,Z 874.943,A -85,B 0,C 180,E1 14626.44,E2 14626.44} C_VEL
LIN {X 0,Y 336.743,Z 857.206,A -85,B 0,C 180,E1 14624.45,E2 14624.45} C_VEL
LIN {X 0,Y 342.332,Z 837.509,A -85,B 0,C 180,E1 14622.656,E2 14622.656} C_VEL
LIN {X 0,Y 347.108,Z 818.467,A -85,B 0,C 180,E1 14621.259,E2 14621.259} C_VEL
LIN {X 0,Y 351.481,Z 798.461,A -85,B 0,C 180,E1 14620.081,E2 14620.081} C_VEL
LIN {X 0,Y 355.111,Z 778.118,A -85,B 0,C 180,E1 14619.171,E2 14619.171} C_VEL
LIN {X 0,Y 358.035,Z 756.302,A -85,B 0,C 180,E1 14618.457,E2 14618.457} C_VEL
LIN {X 0,Y 360.01,Z 730.601,A -85,B 0,C 180,E1 14617.852,E2 14617.852} C_VEL
LIN {X 0,Y 372.237,Z 532.573,A -85,B 0,C 180,E1 14613.728,E2 14613.728} C_VEL
LIN {X 0,Y 365.049,Z 519.186,A -85,B 0,C 180,E1 14611.309,E2 14611.309} C_VEL
LIN {X 0,Y 358.307,Z 508.007,A -85,B 0,C 180,E1 14608.728,E2 14608.728} C_VEL
LIN {X 0,Y 353.394,Z 500.533,A -85,B 0,C 180,E1 14606.553,E2 14606.553} C_VEL
LIN {X 0,Y 350.533,Z 496.29,A -85,B 0,C 180,E1 14605.105,E2 14605.105} C_VEL
LIN {X 0,Y 347.384,Z 491.761,A -85,B 0,C 180,E1 14603.313,E2 14603.313} C_VEL
LIN {X 0,Y 345.174,Z 488.633,A -85,B 0,C 180,E1 14601.852,E2 14601.852} C_VEL
LIN {X 0,Y 341.985,Z 484.101,A -85,B 0,C 180,E1 14599.291,E2 14599.291} C_VEL
LIN {X 0,Y 338.235,Z 479.036,A -85,B 0,C 180,E1 14594.185,E2 14594.185} C_VEL
LIN {X 0,Y 337.541,Z 478.464,A -85,B 0,C 180,E1 14590.237,E2 14590.237} C_VEL
LIN {X 0,Y 338.298,Z 479.318,A -85,B 0,C 180,E1 14587.472,E2 14587.472} C_VEL
LIN {X 0,Y 342.071,Z 484.635,A -85,B 0,C 180,E1 14582.429,E2 14582.429} C_VEL
LIN {X 0,Y 346.04,Z 490.332,A -85,B 0,C 180,E1 14579.337,E2 14579.337} C_VEL
LIN {X 0,Y 349.593,Z 495.572,A -85,B 0,C 180,E1 14577.172,E2 14577.172} C_VEL
LIN {X 0,Y 352.084,Z 499.274,A -85,B 0,C 180,E1 14575.847,E2 14575.847} C_VEL
LIN {X 0,Y 356.704,Z 506.334,A -85,B 0,C 180,E1 14573.683,E2 14573.683} C_VEL
LIN {X 0,Y 363.491,Z 517.63,A -85,B 0,C 180,E1 14570.943,E2 14570.943} C_VEL
LIN {X 0,Y 370.436,Z 530.428,A -85,B 0,C 180,E1 14568.5,E2 14568.5} C_VEL
LIN {X 0,Y 370.803,Z 531.516,A -85,B 0,C 180,E1 14568.364,E2 14568.364} C_VEL
LIN {X 0,Y 356.641,Z 728.609,A -85,B 0,C 180,E1 14564.062,E2 14564.062} C_VEL
LIN {X 0,Y 354.158,Z 749.414,A -85,B 0,C 180,E1 14563.345,E2 14563.345} C_VEL
LIN {X 0,Y 351.011,Z 768.854,A -85,B 0,C 180,E1 14562.425,E2 14562.425} C_VEL
LIN {X 0,Y 346.886,Z 789.282,A -85,B 0,C 180,E1 14561.166,E2 14561.166} C_VEL
LIN {X 0,Y 342.25,Z 808.408,A -85,B 0,C 180,E1 14559.667,E2 14559.667} C_VEL
LIN {X 0,Y 337.091,Z 826.811,A -85,B 0,C 180,E1 14557.87,E2 14557.87} C_VEL
LIN {X 0,Y 331.333,Z 844.932,A -85,B 0,C 180,E1 14555.678,E2 14555.678} C_VEL
LIN {X 0,Y 325.696,Z 861.055,A -85,B 0,C 180,E1 14553.284,E2 14553.284} C_VEL
LIN {X 0,Y 320.152,Z 875.883,A -85,B 0,C 180,E1 14550.603,E2 14550.603} C_VEL
LIN {X 0,Y 314.719,Z 889.841,A -85,B 0,C 180,E1 14547.526,E2 14547.526} C_VEL
LIN {X 0,Y 309.927,Z 901.881,A -85,B 0,C 180,E1 14544.272,E2 14544.272} C_VEL
LIN {X 0,Y 305.807,Z 912.357,A -85,B 0,C 180,E1 14540.787,E2 14540.787} C_VEL
LIN {X 0,Y 302.339,Z 921.556,A -85,B 0,C 180,E1 14536.951,E2 14536.951} C_VEL
LIN {X 0,Y 299.733,Z 929.069,A -85,B 0,C 180,E1 14532.876,E2 14532.876} C_VEL
LIN {X 0,Y 298.064,Z 934.522,A -85,B 0,C 180,E1 14528.844,E2 14528.844} C_VEL
LIN {X 0,Y 297.144,Z 938.18,A -85,B 0,C 180,E1 14524.886,E2 14524.886} C_VEL
LIN {X 0,Y 296.71,Z 940.311,A -85,B 0,C 180,E1 14520.805,E2 14520.805} C_VEL
LIN {X 0,Y 296.592,Z 940.867,A -85,B 0,C 180,E1 14517.066,E2 14517.066} C_VEL
LIN {X 0,Y 296.657,Z 939.905,A -85,B 0,C 180,E1 14513.219,E2 14513.219} C_VEL
LIN {X 0,Y 297.013,Z 937.398,A -85,B 0,C 180,E1 14509.258,E2 14509.258} C_VEL
LIN {X 0,Y 297.787,Z 933.399,A -85,B 0,C 180,E1 14505.377,E2 14505.377} C_VEL
LIN {X 0,Y 299.175,Z 927.876,A -85,B 0,C 180,E1 14501.563,E2 14501.563} C_VEL
LIN {X 0,Y 301.411,Z 920.235,A -85,B 0,C 180,E1 14497.621,E2 14497.621} C_VEL
LIN {X 0,Y 304.366,Z 911.149,A -85,B 0,C 180,E1 14493.952,E2 14493.952} C_VEL
LIN {X 0,Y 307.973,Z 900.689,A -85,B 0,C 180,E1 14490.538,E2 14490.538} C_VEL
LIN {X 0,Y 312.34,Z 888.326,A -85,B 0,C 180,E1 14487.244,E2 14487.244} C_VEL
LIN {X 0,Y 316.888,Z 875.316,A -85,B 0,C 180,E1 14484.383,E2 14484.383} C_VEL
LIN {X 0,Y 322.065,Z 859.982,A -85,B 0,C 180,E1 14481.606,E2 14481.606} C_VEL
LIN {X 0,Y 327.237,Z 843.514,A -85,B 0,C 180,E1 14479.166,E2 14479.166} C_VEL
LIN {X 0,Y 332.067,Z 826.742,A -85,B 0,C 180,E1 14477.122,E2 14477.122} C_VEL
LIN {X 0,Y 336.819,Z 808.448,A -85,B 0,C 180,E1 14475.294,E2 14475.294} C_VEL
LIN {X 0,Y 341.147,Z 789.263,A -85,B 0,C 180,E1 14473.743,E2 14473.743} C_VEL
LIN {X 0,Y 344.855,Z 769.758,A -85,B 0,C 180,E1 14472.491,E2 14472.491} C_VEL
LIN {X 0,Y 348.083,Z 748.515,A -85,B 0,C 180,E1 14471.456,E2 14471.456} C_VEL
LIN {X 0,Y 350.38,Z 727.371,A -85,B 0,C 180,E1 14470.722,E2 14470.722} C_VEL
LIN {X 0,Y 352.716,Z 690.954,A -85,B 0,C 180,E1 14469.894,E2 14469.894} C_VEL
LIN {X 0,Y 353.035,Z 685.437,A -85,B 0,C 180,E1 14469.776,E2 14469.776} C_VEL
LIN {X 0,Y 352.79,Z 677.868,A -85,B 0,C 180,E1 14469.494,E2 14469.494} C_VEL
LIN {X 0,Y 349.765,Z 658.117,A -85,B 0,C 180,E1 14468.313,E2 14468.313} C_VEL
LIN {X 0,Y 349.683,Z 651.608,A -85,B 0,C 180,E1 14468.085,E2 14468.085} C_VEL
LIN {X 0,Y 357.117,Z 529.991,A -85,B 0,C 180,E1 14465.498,E2 14465.498} C_VEL
LIN {X 0,Y 348.14,Z 514.471,A -85,B 0,C 180,E1 14463.046,E2 14463.046} C_VEL
LIN {X 0,Y 337.726,Z 498.106,A -85,B 0,C 180,E1 14459.935,E2 14459.935} C_VEL
LIN {X 0,Y 328.801,Z 485.308,A -85,B 0,C 180,E1 14456.987,E2 14456.987} C_VEL
LIN {X 0,Y 319.777,Z 472.879,A -85,B 0,C 180,E1 14453.624,E2 14453.624} C_VEL
LIN {X 0,Y 314.505,Z 466.27,A -85,B 0,C 180,E1 14451.451,E2 14451.451} C_VEL
LIN {X 0,Y 309.887,Z 460.464,A -85,B 0,C 180,E1 14449.381,E2 14449.381} C_VEL
LIN {X 0,Y 306.143,Z 455.949,A -85,B 0,C 180,E1 14447.572,E2 14447.572} C_VEL
LIN {X 0,Y 303.573,Z 452.335,A -85,B 0,C 180,E1 14445.972,E2 14445.972} C_VEL
LIN {X 0,Y 302.615,Z 450.648,A -85,B 0,C 180,E1 14444.998,E2 14444.998} C_VEL
LIN {X 0,Y 300.49,Z 446.737,A -85,B 0,C 180,E1 14442.658,E2 14442.658} C_VEL
LIN {X 0,Y 297.438,Z 441.569,A -85,B 0,C 180,E1 14438.949,E2 14438.949} C_VEL
LIN {X 0,Y 296.204,Z 439.877,A -85,B 0,C 180,E1 14437.417,E2 14437.417} C_VEL
LIN {X 0,Y 293.576,Z 435.112,A -85,B 0,C 180,E1 14433.02,E2 14433.02} C_VEL
LIN {X 0,Y 290.381,Z 429.764,A -85,B 0,C 180,E1 14424.698,E2 14424.698} C_VEL
LIN {X 0,Y 290.35,Z 429.525,A -85,B 0,C 180,E1 14419.934,E2 14419.934} C_VEL
LIN {X 0,Y 290.354,Z 429.53,A -85,B 0,C 180,E1 14415.368,E2 14415.368} C_VEL
LIN {X 0,Y 290.361,Z 429.623,A -85,B 0,C 180,E1 14410.717,E2 14410.717} C_VEL
LIN {X 0,Y 290.478,Z 430.265,A -85,B 0,C 180,E1 14407.715,E2 14407.715} C_VEL
LIN {X 0,Y 294.045,Z 435.669,A -85,B 0,C 180,E1 14399.806,E2 14399.806} C_VEL
LIN {X 0,Y 296.431,Z 440.076,A -85,B 0,C 180,E1 14395.939,E2 14395.939} C_VEL
LIN {X 0,Y 297.615,Z 441.449,A -85,B 0,C 180,E1 14394.603,E2 14394.603} C_VEL
LIN {X 0,Y 299.833,Z 445.563,A -85,B 0,C 180,E1 14391.756,E2 14391.756} C_VEL
LIN {X 0,Y 300.972,Z 447.12,A -85,B 0,C 180,E1 14390.632,E2 14390.632} C_VEL
LIN {X 0,Y 303.296,Z 451.161,A -85,B 0,C 180,E1 14388.207,E2 14388.207} C_VEL
LIN {X 0,Y 304.225,Z 452.837,A -85,B 0,C 180,E1 14387.28,E2 14387.28} C_VEL
LIN {X 0,Y 306.616,Z 456.258,A -85,B 0,C 180,E1 14385.748,E2 14385.748} C_VEL
LIN {X 0,Y 308.696,Z 458.634,A -85,B 0,C 180,E1 14384.743,E2 14384.743} C_VEL
LIN {X 0,Y 313.204,Z 464.172,A -85,B 0,C 180,E1 14382.634,E2 14382.634} C_VEL
LIN {X 0,Y 317.709,Z 469.809,A -85,B 0,C 180,E1 14380.705,E2 14380.705} C_VEL
LIN {X 0,Y 324.983,Z 479.156,A -85,B 0,C 180,E1 14377.859,E2 14377.859} C_VEL
LIN {X 0,Y 333.409,Z 490.773,A -85,B 0,C 180,E1 14374.891,E2 14374.891} C_VEL
LIN {X 0,Y 342.224,Z 503.488,A -85,B 0,C 180,E1 14372.083,E2 14372.083} C_VEL
LIN {X 0,Y 351.514,Z 517.796,A -85,B 0,C 180,E1 14369.393,E2 14369.393} C_VEL
LIN {X 0,Y 362.008,Z 535.305,A -85,B 0,C 180,E1 14366.613,E2 14366.613} C_VEL
LIN {X 0,Y 349.687,Z 752.141,A -85,B 0,C 180,E1 14362.132,E2 14362.132} C_VEL
LIN {X 0,Y 347.101,Z 774.288,A -85,B 0,C 180,E1 14361.455,E2 14361.455} C_VEL
LIN {X 0,Y 343.697,Z 795.247,A -85,B 0,C 180,E1 14360.571,E2 14360.571} C_VEL
LIN {X 0,Y 339.616,Z 815.725,A -85,B 0,C 180,E1 14359.43,E2 14359.43} C_VEL
LIN {X 0,Y 334.911,Z 835.464,A -85,B 0,C 180,E1 14358.023,E2 14358.023} C_VEL
LIN {X 0,Y 329.702,Z 854.552,A -85,B 0,C 180,E1 14356.329,E2 14356.329} C_VEL
LIN {X 0,Y 323.897,Z 873.748,A -85,B 0,C 180,E1 14354.243,E2 14354.243} C_VEL
LIN {X 0,Y 318.144,Z 891.479,A -85,B 0,C 180,E1 14351.892,E2 14351.892} C_VEL
LIN {X 0,Y 312.413,Z 907.908,A -85,B 0,C 180,E1 14349.241,E2 14349.241} C_VEL
LIN {X 0,Y 307.068,Z 922.843,A -85,B 0,C 180,E1 14346.347,E2 14346.347} C_VEL
LIN {X 0,Y 302.08,Z 936.841,A -85,B 0,C 180,E1 14343.106,E2 14343.106} C_VEL
LIN {X 0,Y 297.677,Z 949.551,A -85,B 0,C 180,E1 14339.548,E2 14339.548} C_VEL
LIN {X 0,Y 294.023,Z 960.883,A -85,B 0,C 180,E1 14335.69,E2 14335.69} C_VEL
LIN {X 0,Y 291.235,Z 970.896,A -85,B 0,C 180,E1 14331.506,E2 14331.506} C_VEL
LIN {X 0,Y 289.538,Z 978.643,A -85,B 0,C 180,E1 14327.488,E2 14327.488} C_VEL
LIN {X 0,Y 288.617,Z 984.647,A -85,B 0,C 180,E1 14323.425,E2 14323.425} C_VEL
LIN {X 0,Y 288.3,Z 989.255,A -85,B 0,C 180,E1 14319.184,E2 14319.184} C_VEL
LIN {X 0,Y 288.334,Z 991.943,A -85,B 0,C 180,E1 14315.376,E2 14315.376} C_VEL
LIN {X 0,Y 288.431,Z 993.188,A -85,B 0,C 180,E1 14311.593,E2 14311.593} C_VEL
LIN {X 0,Y 288.43,Z 993.125,A -85,B 0,C 180,E1 14308.216,E2 14308.216} C_VEL
LIN {X 0,Y 288.335,Z 991.763,A -85,B 0,C 180,E1 14304.395,E2 14304.395} C_VEL
LIN {X 0,Y 288.305,Z 988.968,A -85,B 0,C 180,E1 14300.624,E2 14300.624} C_VEL
LIN {X 0,Y 288.613,Z 984.569,A -85,B 0,C 180,E1 14296.583,E2 14296.583} C_VEL
LIN {X 0,Y 289.528,Z 978.521,A -85,B 0,C 180,E1 14292.521,E2 14292.521} C_VEL
LIN {X 0,Y 291.351,Z 970.355,A -85,B 0,C 180,E1 14288.25,E2 14288.25} C_VEL
LIN {X 0,Y 294.096,Z 960.77,A -85,B 0,C 180,E1 14284.209,E2 14284.209} C_VEL
LIN {X 0,Y 297.934,Z 949.215,A -85,B 0,C 180,E1 14280.225,E2 14280.225} C_VEL
LIN {X 0,Y 302.375,Z 936.789,A -85,B 0,C 180,E1 14276.714,E2 14276.714} C_VEL
LIN {X 0,Y 307.784,Z 922.314,A -85,B 0,C 180,E1 14273.298,E2 14273.298} C_VEL
LIN {X 0,Y 313.621,Z 906.877,A -85,B 0,C 180,E1 14270.273,E2 14270.273} C_VEL
LIN {X 0,Y 319.825,Z 889.925,A -85,B 0,C 180,E1 14267.531,E2 14267.531} C_VEL
LIN {X 0,Y 325.786,Z 872.682,A -85,B 0,C 180,E1 14265.23,E2 14265.23} C_VEL
LIN {X 0,Y 332.006,Z 853.474,A -85,B 0,C 180,E1 14263.127,E2 14263.127} C_VEL
LIN {X 0,Y 337.488,Z 834.867,A -85,B 0,C 180,E1 14261.456,E2 14261.456} C_VEL
LIN {X 0,Y 342.641,Z 814.656,A -85,B 0,C 180,E1 14260.012,E2 14260.012} C_VEL
LIN {X 0,Y 347.191,Z 793.684,A -85,B 0,C 180,E1 14258.839,E2 14258.839} C_VEL
LIN {X 0,Y 350.906,Z 772.747,A -85,B 0,C 180,E1 14257.956,E2 14257.956} C_VEL
LIN {X 0,Y 353.771,Z 750.332,A -85,B 0,C 180,E1 14257.271,E2 14257.271} C_VEL
LIN {X 0,Y 357.911,Z 686.06,A -85,B 0,C 180,E1 14255.894,E2 14255.894} C_VEL
LIN {X 0,Y 367.72,Z 536.375,A -85,B 0,C 180,E1 14252.735,E2 14252.735} C_VEL
LIN {X 0,Y 361.178,Z 524.109,A -85,B 0,C 180,E1 14250.391,E2 14250.391} C_VEL
LIN {X 0,Y 355.054,Z 513.605,A -85,B 0,C 180,E1 14247.87,E2 14247.87} C_VEL
LIN {X 0,Y 349.569,Z 504.997,A -85,B 0,C 180,E1 14245.225,E2 14245.225} C_VEL
LIN {X 0,Y 345.447,Z 498.953,A -85,B 0,C 180,E1 14242.82,E2 14242.82} C_VEL
LIN {X 0,Y 343.561,Z 496.207,A -85,B 0,C 180,E1 14241.511,E2 14241.511} C_VEL
LIN {X 0,Y 340.594,Z 491.829,A -85,B 0,C 180,E1 14239.017,E2 14239.017} C_VEL
LIN {X 0,Y 337.107,Z 486.932,A -85,B 0,C 180,E1 14234.076,E2 14234.076} C_VEL
LIN {X 0,Y 336.477,Z 486.398,A -85,B 0,C 180,E1 14230.097,E2 14230.097} C_VEL
LIN {X 0,Y 337.188,Z 487.308,A -85,B 0,C 180,E1 14227.496,E2 14227.496} C_VEL
LIN {X 0,Y 340.584,Z 492.221,A -85,B 0,C 180,E1 14222.776,E2 14222.776} C_VEL
LIN {X 0,Y 344.378,Z 497.91,A -85,B 0,C 180,E1 14219.667,E2 14219.667} C_VEL
LIN {X 0,Y 349.073,Z 504.86,A -85,B 0,C 180,E1 14216.798,E2 14216.798} C_VEL
LIN {X 0,Y 354.653,Z 513.946,A -85,B 0,C 180,E1 14214.012,E2 14214.012} C_VEL
LIN {X 0,Y 360.81,Z 524.538,A -85,B 0,C 180,E1 14211.433,E2 14211.433} C_VEL
LIN {X 0,Y 366.406,Z 535.236,A -85,B 0,C 180,E1 14209.355,E2 14209.355} C_VEL
LIN {X 0,Y 351.86,Z 729.086,A -85,B 0,C 180,E1 14205.097,E2 14205.097} C_VEL
LIN {X 0,Y 349.291,Z 749.882,A -85,B 0,C 180,E1 14204.379,E2 14204.379} C_VEL
LIN {X 0,Y 346.008,Z 769.488,A -85,B 0,C 180,E1 14203.449,E2 14203.449} C_VEL
LIN {X 0,Y 341.779,Z 789.622,A -85,B 0,C 180,E1 14202.202,E2 14202.202} C_VEL
LIN {X 0,Y 337.233,Z 807.785,A -85,B 0,C 180,E1 14200.785,E2 14200.785} C_VEL
LIN {X 0,Y 331.668,Z 826.894,A -85,B 0,C 180,E1 14198.921,E2 14198.921} C_VEL
LIN {X 0,Y 326.099,Z 843.747,A -85,B 0,C 180,E1 14196.888,E2 14196.888} C_VEL
LIN {X 0,Y 320.158,Z 860.118,A -85,B 0,C 180,E1 14194.483,E2 14194.483} C_VEL
LIN {X 0,Y 314.126,Z 875.652,A -85,B 0,C 180,E1 14191.688,E2 14191.688} C_VEL
LIN {X 0,Y 308.679,Z 888.97,A -85,B 0,C 180,E1 14188.764,E2 14188.764} C_VEL
LIN {X 0,Y 303.571,Z 901.182,A -85,B 0,C 180,E1 14185.492,E2 14185.492} C_VEL
LIN {X 0,Y 298.925,Z 912.262,A -85,B 0,C 180,E1 14181.808,E2 14181.808} C_VEL
LIN {X 0,Y 295.123,Z 921.569,A -85,B 0,C 180,E1 14177.89,E2 14177.89} C_VEL
LIN {X 0,Y 292.369,Z 928.836,A -85,B 0,C 180,E1 14173.958,E2 14173.958} C_VEL
LIN {X 0,Y 290.436,Z 934.581,A -85,B 0,C 180,E1 14169.809,E2 14169.809} C_VEL
LIN {X 0,Y 289.332,Z 938.524,A -85,B 0,C 180,E1 14165.697,E2 14165.697} C_VEL
LIN {X 0,Y 288.824,Z 940.819,A -85,B 0,C 180,E1 14161.743,E2 14161.743} C_VEL
LIN {X 0,Y 288.632,Z 941.552,A -85,B 0,C 180,E1 14157.877,E2 14157.877} C_VEL
LIN {X 0,Y 288.664,Z 940.883,A -85,B 0,C 180,E1 14153.874,E2 14153.874} C_VEL
LIN {X 0,Y 288.962,Z 938.87,A -85,B 0,C 180,E1 14150.028,E2 14150.028} C_VEL
LIN {X 0,Y 289.665,Z 935.2,A -85,B 0,C 180,E1 14146.025,E2 14146.025} C_VEL
LIN {X 0,Y 290.969,Z 929.974,A -85,B 0,C 180,E1 14142.095,E2 14142.095} C_VEL
LIN {X 0,Y 293.151,Z 922.762,A -85,B 0,C 180,E1 14138.034,E2 14138.034} C_VEL
LIN {X 0,Y 296.08,Z 914.148,A -85,B 0,C 180,E1 14134.256,E2 14134.256} C_VEL
LIN {X 0,Y 299.671,Z 904.253,A -85,B 0,C 180,E1 14130.761,E2 14130.761} C_VEL
LIN {X 0,Y 304.329,Z 891.669,A -85,B 0,C 180,E1 14127.18,E2 14127.18} C_VEL
LIN {X 0,Y 309.267,Z 878.131,A -85,B 0,C 180,E1 14124.058,E2 14124.058} C_VEL
LIN {X 0,Y 314.38,Z 863.631,A -85,B 0,C 180,E1 14121.307,E2 14121.307} C_VEL
LIN {X 0,Y 319.678,Z 847.724,A -85,B 0,C 180,E1 14118.815,E2 14118.815} C_VEL
LIN {X 0,Y 325.031,Z 830.241,A -85,B 0,C 180,E1 14116.567,E2 14116.567} C_VEL
LIN {X 0,Y 329.932,Z 812.565,A -85,B 0,C 180,E1 14114.71,E2 14114.71} C_VEL
LIN {X 0,Y 334.615,Z 793.122,A -85,B 0,C 180,E1 14113.059,E2 14113.059} C_VEL
LIN {X 0,Y 338.732,Z 772.507,A -85,B 0,C 180,E1 14111.684,E2 14111.684} C_VEL
LIN {X 0,Y 342.015,Z 752.024,A -85,B 0,C 180,E1 14110.646,E2 14110.646} C_VEL
LIN {X 0,Y 344.523,Z 731.073,A -85,B 0,C 180,E1 14109.871,E2 14109.871} C_VEL
LIN {X 0,Y 346.572,Z 703.152,A -85,B 0,C 180,E1 14109.188,E2 14109.188} C_VEL
LIN {X 0,Y 349.683,Z 651.608,A -85,B 0,C 180,E1 14108.085,E2 14108.085} C_VEL
LIN {X 0,Y 349.51,Z 644.04,A -85,B 0,C 180,E1 14107.803,E2 14107.803} C_VEL
LIN {X 0,Y 346.667,Z 624.305,A -85,B 0,C 180,E1 14106.592,E2 14106.592} C_VEL
LIN {X 0,Y 346.591,Z 617.799,A -85,B 0,C 180,E1 14106.355,E2 14106.355} C_VEL
LIN {X 0,Y 351.972,Z 533.592,A -85,B 0,C 180,E1 14104.556,E2 14104.556} C_VEL
LIN {X 0,Y 342.119,Z 516.688,A -85,B 0,C 180,E1 14101.738,E2 14101.738} C_VEL
LIN {X 0,Y 332.938,Z 502.319,A -85,B 0,C 180,E1 14098.86,E2 14098.86} C_VEL
LIN {X 0,Y 323.592,Z 488.698,A -85,B 0,C 180,E1 14095.589,E2 14095.589} C_VEL
LIN {X 0,Y 316.033,Z 478.587,A -85,B 0,C 180,E1 14092.647,E2 14092.647} C_VEL
LIN {X 0,Y 312.14,Z 473.445,A -85,B 0,C 180,E1 14090.968,E2 14090.968} C_VEL
LIN {X 0,Y 307.146,Z 467.138,A -85,B 0,C 180,E1 14088.674,E2 14088.674} C_VEL
LIN {X 0,Y 303.858,Z 463.087,A -85,B 0,C 180,E1 14087.02,E2 14087.02} C_VEL
